LIN {X 0,Y 418.354,Z 136.374,A -85,B 0,C 180,E1 -10247.385,E2 -10247.385} C_VEL
LIN {X 0,Y 418.34,Z 136.372,A -85,B 0,C 180,E1 -10250.328,E2 -10250.328} C_VEL
LIN {X 0,Y 418.511,Z 136.347,A -85,B 0,C 180,E1 -10252.279,E2 -10252.279} C_VEL
LIN {X 0,Y 418.512,Z 136.351,A -85,B 0,C 180,E1 -10254.217,E2 -10254.217} C_VEL
LIN {X 0,Y 418.543,Z 136.347,A -85,B 0,C 180,E1 -10258.075,E2 -10258.075} C_VEL
LIN {X 0,Y 418.671,Z 136.328,A -85,B 0,C 180,E1 -10260,E2 -10260} C_VEL
LIN {X 0,Y 418.508,Z 136.353,A -85,B 0,C 180,E1 -10262.888,E2 -10262.888} C_VEL
LIN {X 0,Y 418.485,Z 136.356,A -85,B 0,C 180,E1 -10266.751,E2 -10266.751} C_VEL
LIN {X 0,Y 418.339,Z 136.373,A -85,B 0,C 180,E1 -10269.671,E2 -10269.671} C_VEL
LIN {X 0,Y 418.344,Z 136.376,A -85,B 0,C 180,E1 -10273.001,E2 -10273.001} C_VEL
LIN {X 0,Y 418.311,Z 136.381,A -85,B 0,C 180,E1 -10276.735,E2 -10276.735} C_VEL
LIN {X 0,Y 418.269,Z 136.382,A -85,B 0,C 180,E1 -10279.79,E2 -10279.79} C_VEL
LIN {X 0,Y 418.236,Z 136.392,A -85,B 0,C 180,E1 -10282.736,E2 -10282.736} C_VEL
LIN {X 0,Y 418.268,Z 136.387,A -85,B 0,C 180,E1 -10285.904,E2 -10285.904} C_VEL
LIN {X 0,Y 418.262,Z 136.385,A -85,B 0,C 180,E1 -10289.162,E2 -10289.162} C_VEL
LIN {X 0,Y 418.279,Z 136.588,A -85,B 0,C 180,E1 -10291.885,E2 -10291.885} C_VEL
LIN {X 0,Y 419.996,Z 144.56,A -85,B 0,C 180,E1 -10293.806,E2 -10293.806} C_VEL
LIN {X 0,Y 422.177,Z 151.711,A -85,B 0,C 180,E1 -10294.075,E2 -10294.075} C_VEL
LIN {X 0,Y 424.507,Z 162.243,A -85,B 0,C 180,E1 -10294.391,E2 -10294.391} C_VEL
LIN {X 0,Y 423.252,Z 251.811,A -85,B 0,C 180,E1 -10296.015,E2 -10296.015} C_VEL
LIN {X 0,Y 422.853,Z 265.002,A -85,B 0,C 180,E1 -10296.445,E2 -10296.445} C_VEL
LIN {X 0,Y 422.454,Z 276.75,A -85,B 0,C 180,E1 -10297.01,E2 -10297.01} C_VEL
LIN {X 0,Y 421.875,Z 288.685,A -85,B 0,C 180,E1 -10297.778,E2 -10297.778} C_VEL
LIN {X 0,Y 421.216,Z 299.793,A -85,B 0,C 180,E1 -10298.706,E2 -10298.706} C_VEL
LIN {X 0,Y 420.478,Z 309.867,A -85,B 0,C 180,E1 -10299.749,E2 -10299.749} C_VEL
LIN {X 0,Y 419.822,Z 318.462,A -85,B 0,C 180,E1 -10300.838,E2 -10300.838} C_VEL
LIN {X 0,Y 419.17,Z 326.786,A -85,B 0,C 180,E1 -10302.118,E2 -10302.118} C_VEL
LIN {X 0,Y 418.53,Z 334.126,A -85,B 0,C 180,E1 -10303.509,E2 -10303.509} C_VEL
LIN {X 0,Y 418.044,Z 340.71,A -85,B 0,C 180,E1 -10305.083,E2 -10305.083} C_VEL
LIN {X 0,Y 417.75,Z 345.057,A -85,B 0,C 180,E1 -10306.389,E2 -10306.389} C_VEL
LIN {X 0,Y 417.461,Z 348.727,A -85,B 0,C 180,E1 -10307.795,E2 -10307.795} C_VEL
LIN {X 0,Y 417.221,Z 351.572,A -85,B 0,C 180,E1 -10309.289,E2 -10309.289} C_VEL
LIN {X 0,Y 417.092,Z 353.429,A -85,B 0,C 180,E1 -10310.814,E2 -10310.814} C_VEL
LIN {X 0,Y 417.018,Z 354.326,A -85,B 0,C 180,E1 -10312.649,E2 -10312.649} C_VEL
LIN {X 0,Y 417.039,Z 354.081,A -85,B 0,C 180,E1 -10313.989,E2 -10313.989} C_VEL
LIN {X 0,Y 417.104,Z 352.704,A -85,B 0,C 180,E1 -10315.652,E2 -10315.652} C_VEL
LIN {X 0,Y 417.278,Z 349.985,A -85,B 0,C 180,E1 -10317.387,E2 -10317.387} C_VEL
LIN {X 0,Y 417.563,Z 345.808,A -85,B 0,C 180,E1 -10319.135,E2 -10319.135} C_VEL
LIN {X 0,Y 417.947,Z 340.265,A -85,B 0,C 180,E1 -10320.814,E2 -10320.814} C_VEL
LIN {X 0,Y 418.428,Z 333.293,A -85,B 0,C 180,E1 -10322.444,E2 -10322.444} C_VEL
LIN {X 0,Y 418.96,Z 325.522,A -85,B 0,C 180,E1 -10323.875,E2 -10323.875} C_VEL
LIN {X 0,Y 419.599,Z 316.285,A -85,B 0,C 180,E1 -10325.246,E2 -10325.246} C_VEL
LIN {X 0,Y 420.213,Z 307.278,A -85,B 0,C 180,E1 -10326.335,E2 -10326.335} C_VEL
LIN {X 0,Y 420.843,Z 297.324,A -85,B 0,C 180,E1 -10327.321,E2 -10327.321} C_VEL
LIN {X 0,Y 421.442,Z 285.916,A -85,B 0,C 180,E1 -10328.22,E2 -10328.22} C_VEL
LIN {X 0,Y 421.997,Z 273.068,A -85,B 0,C 180,E1 -10328.997,E2 -10328.997} C_VEL
LIN {X 0,Y 422.427,Z 260.281,A -85,B 0,C 180,E1 -10329.551,E2 -10329.551} C_VEL
LIN {X 0,Y 422.746,Z 246.227,A -85,B 0,C 180,E1 -10329.932,E2 -10329.932} C_VEL
LIN {X 0,Y 423.437,Z 190.42,A -85,B 0,C 180,E1 -10330.915,E2 -10330.915} C_VEL
LIN {X 0,Y 422.55,Z 182.716,A -85,B 0,C 180,E1 -10331.093,E2 -10331.093} C_VEL
LIN {X 0,Y 418.279,Z 167.8,A -85,B 0,C 180,E1 -10331.551,E2 -10331.551} C_VEL
LIN {X 0,Y 416.448,Z 160.229,A -85,B 0,C 180,E1 -10331.772,E2 -10331.772} C_VEL
LIN {X 0,Y 413.37,Z 146.655,A -85,B 0,C 180,E1 -10332.164,E2 -10332.164} C_VEL
LIN {X 0,Y 412.534,Z 143.848,A -85,B 0,C 180,E1 -10332.276,E2 -10332.276} C_VEL
LIN {X 0,Y 411.31,Z 137.253,A -85,B 0,C 180,E1 -10333.879,E2 -10333.879} C_VEL
LIN {X 0,Y 411.303,Z 137.253,A -85,B 0,C 180,E1 -10337.166,E2 -10337.166} C_VEL
LIN {X 0,Y 411.292,Z 137.25,A -85,B 0,C 180,E1 -10340.161,E2 -10340.161} C_VEL
LIN {X 0,Y 411.452,Z 137.232,A -85,B 0,C 180,E1 -10343.133,E2 -10343.133} C_VEL
LIN {X 0,Y 411.308,Z 137.25,A -85,B 0,C 180,E1 -10345.099,E2 -10345.099} C_VEL
LIN {X 0,Y 411.51,Z 137.222,A -85,B 0,C 180,E1 -10348.043,E2 -10348.043} C_VEL
LIN {X 0,Y 411.64,Z 137.206,A -85,B 0,C 180,E1 -10350,E2 -10350} C_VEL
LIN {X 0,Y 411.457,Z 137.231,A -85,B 0,C 180,E1 -10352.937,E2 -10352.937} C_VEL
LIN {X 0,Y 411.424,Z 137.236,A -85,B 0,C 180,E1 -10356.868,E2 -10356.868} C_VEL
LIN {X 0,Y 411.291,Z 137.249,A -85,B 0,C 180,E1 -10359.839,E2 -10359.839} C_VEL
LIN {X 0,Y 411.305,Z 137.253,A -85,B 0,C 180,E1 -10363.104,E2 -10363.104} C_VEL
LIN {X 0,Y 411.257,Z 137.26,A -85,B 0,C 180,E1 -10366.889,E2 -10366.889} C_VEL
LIN {X 0,Y 411.23,Z 137.257,A -85,B 0,C 180,E1 -10369.987,E2 -10369.987} C_VEL
LIN {X 0,Y 411.196,Z 137.264,A -85,B 0,C 180,E1 -10373.148,E2 -10373.148} C_VEL
LIN {X 0,Y 411.236,Z 137.259,A -85,B 0,C 180,E1 -10376.381,E2 -10376.381} C_VEL
LIN {X 0,Y 411.199,Z 137.26,A -85,B 0,C 180,E1 -10379.713,E2 -10379.713} C_VEL
LIN {X 0,Y 411.205,Z 137.261,A -85,B 0,C 180,E1 -10383.156,E2 -10383.156} C_VEL
LIN {X 0,Y 411.191,Z 137.267,A -85,B 0,C 180,E1 -10386.552,E2 -10386.552} C_VEL
LIN {X 0,Y 411.207,Z 137.26,A -85,B 0,C 180,E1 -10389.727,E2 -10389.727} C_VEL
LIN {X 0,Y 411.172,Z 137.264,A -85,B 0,C 180,E1 -10393.134,E2 -10393.134} C_VEL
LIN {X 0,Y 411.168,Z 137.268,A -85,B 0,C 180,E1 -10395.881,E2 -10395.881} C_VEL
LIN {X 0,Y 411.163,Z 137.266,A -85,B 0,C 180,E1 -10398.771,E2 -10398.771} C_VEL
LIN {X 0,Y 411.21,Z 137.263,A -85,B 0,C 180,E1 -10401.83,E2 -10401.83} C_VEL
LIN {X 0,Y 411.209,Z 137.259,A -85,B 0,C 180,E1 -10405.121,E2 -10405.121} C_VEL
LIN {X 0,Y 411.164,Z 137.271,A -85,B 0,C 180,E1 -10408.003,E2 -10408.003} C_VEL
LIN {X 0,Y 411.216,Z 137.261,A -85,B 0,C 180,E1 -10411.41,E2 -10411.41} C_VEL
LIN {X 0,Y 411.235,Z 137.261,A -85,B 0,C 180,E1 -10413.619,E2 -10413.619} C_VEL
LIN {X 0,Y 411.194,Z 137.261,A -85,B 0,C 180,E1 -10416.852,E2 -10416.852} C_VEL
LIN {X 0,Y 411.213,Z 137.261,A -85,B 0,C 180,E1 -10420.05,E2 -10420.05} C_VEL
LIN {X 0,Y 411.261,Z 137.255,A -85,B 0,C 180,E1 -10423.131,E2 -10423.131} C_VEL
LIN {X 0,Y 411.304,Z 137.249,A -85,B 0,C 180,E1 -10426.896,E2 -10426.896} C_VEL
LIN {X 0,Y 411.292,Z 137.249,A -85,B 0,C 180,E1 -10430.161,E2 -10430.161} C_VEL
LIN {X 0,Y 411.459,Z 137.233,A -85,B 0,C 180,E1 -10433.133,E2 -10433.133} C_VEL
LIN {X 0,Y 411.31,Z 137.252,A -85,B 0,C 180,E1 -10435.099,E2 -10435.099} C_VEL
LIN {X 0,Y 411.512,Z 137.221,A -85,B 0,C 180,E1 -10438.043,E2 -10438.043} C_VEL
LIN {X 0,Y 411.641,Z 137.205,A -85,B 0,C 180,E1 -10440,E2 -10440} C_VEL
LIN {X 0,Y 411.464,Z 137.233,A -85,B 0,C 180,E1 -10442.937,E2 -10442.937} C_VEL
LIN {X 0,Y 411.45,Z 137.235,A -85,B 0,C 180,E1 -10446.867,E2 -10446.867} C_VEL
LIN {X 0,Y 411.292,Z 137.249,A -85,B 0,C 180,E1 -10449.839,E2 -10449.839} C_VEL
LIN {X 0,Y 411.304,Z 137.251,A -85,B 0,C 180,E1 -10453.104,E2 -10453.104} C_VEL
LIN {X 0,Y 411.256,Z 137.258,A -85,B 0,C 180,E1 -10456.889,E2 -10456.889} C_VEL
LIN {X 0,Y 411.23,Z 137.258,A -85,B 0,C 180,E1 -10459.987,E2 -10459.987} C_VEL
LIN {X 0,Y 411.196,Z 137.262,A -85,B 0,C 180,E1 -10463.148,E2 -10463.148} C_VEL
LIN {X 0,Y 411.237,Z 137.262,A -85,B 0,C 180,E1 -10466.381,E2 -10466.381} C_VEL
LIN {X 0,Y 411.2,Z 137.261,A -85,B 0,C 180,E1 -10469.713,E2 -10469.713} C_VEL
LIN {X 0,Y 411.206,Z 137.26,A -85,B 0,C 180,E1 -10473.156,E2 -10473.156} C_VEL
LIN {X 0,Y 411.195,Z 137.264,A -85,B 0,C 180,E1 -10476.553,E2 -10476.553} C_VEL
LIN {X 0,Y 411.227,Z 137.26,A -85,B 0,C 180,E1 -10479.731,E2 -10479.731} C_VEL
LIN {X 0,Y 411.178,Z 137.263,A -85,B 0,C 180,E1 -10483.133,E2 -10483.133} C_VEL
LIN {X 0,Y 411.169,Z 137.27,A -85,B 0,C 180,E1 -10485.881,E2 -10485.881} C_VEL
LIN {X 0,Y 411.201,Z 137.26,A -85,B 0,C 180,E1 -10488.766,E2 -10488.766} C_VEL
LIN {X 0,Y 411.205,Z 137.264,A -85,B 0,C 180,E1 -10492.028,E2 -10492.028} C_VEL
LIN {X 0,Y 411.208,Z 137.266,A -85,B 0,C 180,E1 -10495.667,E2 -10495.667} C_VEL
LIN {X 0,Y 411.191,Z 137.264,A -85,B 0,C 180,E1 -10499.153,E2 -10499.153} C_VEL
LIN {X 0,Y 411.287,Z 137.341,A -85,B 0,C 180,E1 -10501.234,E2 -10501.234} C_VEL
LIN {X 0,Y 413.809,Z 149.635,A -85,B 0,C 180,E1 -10503.796,E2 -10503.796} C_VEL
LIN {X 0,Y 414.551,Z 154.098,A -85,B 0,C 180,E1 -10504.698,E2 -10504.698} C_VEL
LIN {X 0,Y 413.345,Z 171.886,A -85,B 0,C 180,E1 -10508.034,E2 -10508.034} C_VEL
LIN {X 0,Y 412.497,Z 186.557,A -85,B 0,C 180,E1 -10510.757,E2 -10510.757} C_VEL
LIN {X 0,Y 416.517,Z 216.408,A -85,B 0,C 180,E1 -10511.49,E2 -10511.49} C_VEL
LIN {X 0,Y 415.495,Z 295.911,A -85,B 0,C 180,E1 -10512.941,E2 -10512.941} C_VEL
LIN {X 0,Y 414.943,Z 309.622,A -85,B 0,C 180,E1 -10513.392,E2 -10513.392} C_VEL
LIN {X 0,Y 414.318,Z 322.023,A -85,B 0,C 180,E1 -10514,E2 -10514} C_VEL
LIN {X 0,Y 413.48,Z 334.717,A -85,B 0,C 180,E1 -10514.851,E2 -10514.851} C_VEL
LIN {X 0,Y 412.731,Z 346.038,A -85,B 0,C 180,E1 -10515.831,E2 -10515.831} C_VEL
LIN {X 0,Y 411.983,Z 356.552,A -85,B 0,C 180,E1 -10516.977,E2 -10516.977} C_VEL
LIN {X 0,Y 411.43,Z 365.442,A -85,B 0,C 180,E1 -10518.172,E2 -10518.172} C_VEL
LIN {X 0,Y 410.734,Z 374.404,A -85,B 0,C 180,E1 -10519.65,E2 -10519.65} C_VEL
LIN {X 0,Y 410.366,Z 381.605,A -85,B 0,C 180,E1 -10521.133,E2 -10521.133} C_VEL
LIN {X 0,Y 410.171,Z 387.34,A -85,B 0,C 180,E1 -10522.617,E2 -10522.617} C_VEL
LIN {X 0,Y 410.003,Z 391.842,A -85,B 0,C 180,E1 -10524.097,E2 -10524.097} C_VEL
LIN {X 0,Y 410.066,Z 394.22,A -85,B 0,C 180,E1 -10525.084,E2 -10525.084} C_VEL
LIN {X 0,Y 409.974,Z 396.148,A -85,B 0,C 180,E1 -10526.068,E2 -10526.068} C_VEL
LIN {X 0,Y 410.06,Z 397.644,A -85,B 0,C 180,E1 -10527.053,E2 -10527.053} C_VEL
LIN {X 0,Y 410.053,Z 398.68,A -85,B 0,C 180,E1 -10528.036,E2 -10528.036} C_VEL
LIN {X 0,Y 410.033,Z 399.317,A -85,B 0,C 180,E1 -10529.018,E2 -10529.018} C_VEL
LIN {X 0,Y 410.034,Z 399.56,A -85,B 0,C 180,E1 -10530,E2 -10530} C_VEL
LIN {X 0,Y 410.02,Z 399.386,A -85,B 0,C 180,E1 -10530.982,E2 -10530.982} C_VEL
LIN {X 0,Y 410.044,Z 398.781,A -85,B 0,C 180,E1 -10531.964,E2 -10531.964} C_VEL
LIN {X 0,Y 410.029,Z 397.777,A -85,B 0,C 180,E1 -10532.947,E2 -10532.947} C_VEL
LIN {X 0,Y 409.972,Z 396.368,A -85,B 0,C 180,E1 -10533.932,E2 -10533.932} C_VEL
LIN {X 0,Y 410.017,Z 393.411,A -85,B 0,C 180,E1 -10535.409,E2 -10535.409} C_VEL
LIN {X 0,Y 410.078,Z 389.406,A -85,B 0,C 180,E1 -10536.89,E2 -10536.89} C_VEL
LIN {X 0,Y 410.357,Z 383.275,A -85,B 0,C 180,E1 -10538.619,E2 -10538.619} C_VEL
LIN {X 0,Y 410.711,Z 376.554,A -85,B 0,C 180,E1 -10540.102,E2 -10540.102} C_VEL
LIN {X 0,Y 411.339,Z 368.229,A -85,B 0,C 180,E1 -10541.581,E2 -10541.581} C_VEL
LIN {X 0,Y 411.91,Z 359.73,A -85,B 0,C 180,E1 -10542.815,E2 -10542.815} C_VEL
LIN {X 0,Y 412.688,Z 349.532,A -85,B 0,C 180,E1 -10544.019,E2 -10544.019} C_VEL
LIN {X 0,Y 413.565,Z 337.56,A -85,B 0,C 180,E1 -10545.146,E2 -10545.146} C_VEL
LIN {X 0,Y 414.45,Z 325.957,A -85,B 0,C 180,E1 -10545.995,E2 -10545.995} C_VEL
LIN {X 0,Y 415.255,Z 312.671,A -85,B 0,C 180,E1 -10546.721,E2 -10546.721} C_VEL
LIN {X 0,Y 415.952,Z 299.229,A -85,B 0,C 180,E1 -10547.23,E2 -10547.23} C_VEL
LIN {X 0,Y 416.316,Z 284.215,A -85,B 0,C 180,E1 -10547.563,E2 -10547.563} C_VEL
LIN {X 0,Y 417.118,Z 215.058,A -85,B 0,C 180,E1 -10548.823,E2 -10548.823} C_VEL
LIN {X 0,Y 414.02,Z 193.054,A -85,B 0,C 180,E1 -10549.4,E2 -10549.4} C_VEL
LIN {X 0,Y 412.69,Z 185.111,A -85,B 0,C 180,E1 -10549.628,E2 -10549.628} C_VEL
LIN {X 0,Y 413.943,Z 164.842,A -85,B 0,C 180,E1 -10553.381,E2 -10553.381} C_VEL
LIN {X 0,Y 414.609,Z 153.401,A -85,B 0,C 180,E1 -10555.534,E2 -10555.534} C_VEL
LIN {X 0,Y 412.265,Z 141.515,A -85,B 0,C 180,E1 -10558.008,E2 -10558.008} C_VEL
LIN {X 0,Y 411.236,Z 137.263,A -85,B 0,C 180,E1 -10558.951,E2 -10558.951} C_VEL
LIN {X 0,Y 411.167,Z 137.271,A -85,B 0,C 180,E1 -10561.997,E2 -10561.997} C_VEL
LIN {X 0,Y 411.212,Z 137.264,A -85,B 0,C 180,E1 -10564.878,E2 -10564.878} C_VEL
LIN {X 0,Y 411.215,Z 137.27,A -85,B 0,C 180,E1 -10568.17,E2 -10568.17} C_VEL
LIN {X 0,Y 411.201,Z 137.264,A -85,B 0,C 180,E1 -10571.234,E2 -10571.234} C_VEL
LIN {X 0,Y 411.176,Z 137.27,A -85,B 0,C 180,E1 -10574.49,E2 -10574.49} C_VEL
LIN {X 0,Y 411.198,Z 137.264,A -85,B 0,C 180,E1 -10578.197,E2 -10578.197} C_VEL
LIN {X 0,Y 411.23,Z 137.256,A -85,B 0,C 180,E1 -10580.777,E2 -10580.777} C_VEL
LIN {X 0,Y 411.198,Z 137.262,A -85,B 0,C 180,E1 -10584.471,E2 -10584.471} C_VEL
LIN {X 0,Y 411.206,Z 137.258,A -85,B 0,C 180,E1 -10586.873,E2 -10586.873} C_VEL
LIN {X 0,Y 411.232,Z 137.253,A -85,B 0,C 180,E1 -10590.644,E2 -10590.644} C_VEL
LIN {X 0,Y 411.235,Z 137.257,A -85,B 0,C 180,E1 -10593.619,E2 -10593.619} C_VEL
LIN {X 0,Y 411.194,Z 137.26,A -85,B 0,C 180,E1 -10596.852,E2 -10596.852} C_VEL
LIN {X 0,Y 411.214,Z 137.257,A -85,B 0,C 180,E1 -10600.05,E2 -10600.05} C_VEL
LIN {X 0,Y 411.262,Z 137.255,A -85,B 0,C 180,E1 -10603.131,E2 -10603.131} C_VEL
LIN {X 0,Y 411.304,Z 137.25,A -85,B 0,C 180,E1 -10606.896,E2 -10606.896} C_VEL
LIN {X 0,Y 411.292,Z 137.25,A -85,B 0,C 180,E1 -10610.161,E2 -10610.161} C_VEL
LIN {X 0,Y 411.459,Z 137.229,A -85,B 0,C 180,E1 -10613.133,E2 -10613.133} C_VEL
LIN {X 0,Y 411.309,Z 137.251,A -85,B 0,C 180,E1 -10615.099,E2 -10615.099} C_VEL
LIN {X 0,Y 411.512,Z 137.223,A -85,B 0,C 180,E1 -10618.042,E2 -10618.042} C_VEL
LIN {X 0,Y 411.64,Z 137.204,A -85,B 0,C 180,E1 -10620,E2 -10620} C_VEL
LIN {X 0,Y 411.463,Z 137.23,A -85,B 0,C 180,E1 -10622.937,E2 -10622.937} C_VEL
LIN {X 0,Y 411.449,Z 137.233,A -85,B 0,C 180,E1 -10626.867,E2 -10626.867} C_VEL
LIN {X 0,Y 411.291,Z 137.251,A -85,B 0,C 180,E1 -10629.839,E2 -10629.839} C_VEL
LIN {X 0,Y 411.303,Z 137.252,A -85,B 0,C 180,E1 -10633.104,E2 -10633.104} C_VEL
LIN {X 0,Y 411.255,Z 137.26,A -85,B 0,C 180,E1 -10636.889,E2 -10636.889} C_VEL
LIN {X 0,Y 411.228,Z 137.26,A -85,B 0,C 180,E1 -10639.987,E2 -10639.987} C_VEL
LIN {X 0,Y 411.201,Z 137.268,A -85,B 0,C 180,E1 -10643.147,E2 -10643.147} C_VEL
LIN {X 0,Y 411.236,Z 137.262,A -85,B 0,C 180,E1 -10646.381,E2 -10646.381} C_VEL
LIN {X 0,Y 411.198,Z 137.264,A -85,B 0,C 180,E1 -10649.713,E2 -10649.713} C_VEL
LIN {X 0,Y 411.218,Z 137.294,A -85,B 0,C 180,E1 -10651.542,E2 -10651.542} C_VEL
LIN {X 0,Y 412.89,Z 145.086,A -85,B 0,C 180,E1 -10653.449,E2 -10653.449} C_VEL
LIN {X 0,Y 415.599,Z 153.137,A -85,B 0,C 180,E1 -10653.754,E2 -10653.754} C_VEL
LIN {X 0,Y 417.868,Z 163.527,A -85,B 0,C 180,E1 -10654.075,E2 -10654.075} C_VEL
LIN {X 0,Y 416.551,Z 251.828,A -85,B 0,C 180,E1 -10655.699,E2 -10655.699} C_VEL
LIN {X 0,Y 416.127,Z 264.942,A -85,B 0,C 180,E1 -10656.127,E2 -10656.127} C_VEL
LIN {X 0,Y 415.704,Z 277.323,A -85,B 0,C 180,E1 -10656.731,E2 -10656.731} C_VEL
LIN {X 0,Y 415.119,Z 288.673,A -85,B 0,C 180,E1 -10657.469,E2 -10657.469} C_VEL
LIN {X 0,Y 414.391,Z 300.39,A -85,B 0,C 180,E1 -10658.462,E2 -10658.462} C_VEL
LIN {X 0,Y 413.545,Z 311.341,A -85,B 0,C 180,E1 -10659.628,E2 -10659.628} C_VEL
LIN {X 0,Y 412.763,Z 321.03,A -85,B 0,C 180,E1 -10660.926,E2 -10660.926} C_VEL
LIN {X 0,Y 411.924,Z 330.134,A -85,B 0,C 180,E1 -10662.447,E2 -10662.447} C_VEL
LIN {X 0,Y 411.396,Z 336.955,A -85,B 0,C 180,E1 -10663.873,E2 -10663.873} C_VEL
LIN {X 0,Y 410.886,Z 343.002,A -85,B 0,C 180,E1 -10665.47,E2 -10665.47} C_VEL
LIN {X 0,Y 410.609,Z 346.964,A -85,B 0,C 180,E1 -10666.793,E2 -10666.793} C_VEL
LIN {X 0,Y 410.352,Z 349.984,A -85,B 0,C 180,E1 -10668.092,E2 -10668.092} C_VEL
LIN {X 0,Y 410.128,Z 352.203,A -85,B 0,C 180,E1 -10669.37,E2 -10669.37} C_VEL
LIN {X 0,Y 410.036,Z 353.731,A -85,B 0,C 180,E1 -10670.641,E2 -10670.641} C_VEL
LIN {X 0,Y 409.945,Z 354.612,A -85,B 0,C 180,E1 -10672.056,E2 -10672.056} C_VEL
LIN {X 0,Y 409.94,Z 354.611,A -85,B 0,C 180,E1 -10673.684,E2 -10673.684} C_VEL
LIN {X 0,Y 410.014,Z 353.235,A -85,B 0,C 180,E1 -10675.553,E2 -10675.553} C_VEL
LIN {X 0,Y 410.139,Z 350.993,A -85,B 0,C 180,E1 -10677.103,E2 -10677.103} C_VEL
LIN {X 0,Y 410.466,Z 347.088,A -85,B 0,C 180,E1 -10678.881,E2 -10678.881} C_VEL
LIN {X 0,Y 410.717,Z 343.026,A -85,B 0,C 180,E1 -10680.249,E2 -10680.249} C_VEL
LIN {X 0,Y 411.164,Z 336.503,A -85,B 0,C 180,E1 -10681.962,E2 -10681.962} C_VEL
LIN {X 0,Y 411.668,Z 329.487,A -85,B 0,C 180,E1 -10683.404,E2 -10683.404} C_VEL
LIN {X 0,Y 412.306,Z 321.233,A -85,B 0,C 180,E1 -10684.777,E2 -10684.777} C_VEL
LIN {X 0,Y 413.039,Z 311.369,A -85,B 0,C 180,E1 -10686.108,E2 -10686.108} C_VEL
LIN {X 0,Y 413.743,Z 300.579,A -85,B 0,C 180,E1 -10687.267,E2 -10687.267} C_VEL
LIN {X 0,Y 414.469,Z 288.693,A -85,B 0,C 180,E1 -10688.278,E2 -10688.278} C_VEL
LIN {X 0,Y 415.002,Z 277.283,A -85,B 0,C 180,E1 -10689.033,E2 -10689.033} C_VEL
LIN {X 0,Y 415.491,Z 264.693,A -85,B 0,C 180,E1 -10689.647,E2 -10689.647} C_VEL
LIN {X 0,Y 415.811,Z 251.596,A -85,B 0,C 180,E1 -10690.082,E2 -10690.082} C_VEL
LIN {X 0,Y 416.955,Z 162.535,A -85,B 0,C 180,E1 -10691.707,E2 -10691.707} C_VEL
LIN {X 0,Y 416.448,Z 160.229,A -85,B 0,C 180,E1 -10691.772,E2 -10691.772} C_VEL
LIN {X 0,Y 415.218,Z 156.314,A -85,B 0,C 180,E1 -10691.914,E2 -10691.914} C_VEL
LIN {X 0,Y 412.319,Z 151.696,A -85,B 0,C 180,E1 -10692.132,E2 -10692.132} C_VEL
LIN {X 0,Y 406.058,Z 144.867,A -85,B 0,C 180,E1 -10692.558,E2 -10692.558} C_VEL
LIN {X 0,Y 405.256,Z 143.561,A -85,B 0,C 180,E1 -10692.76,E2 -10692.76} C_VEL
LIN {X 0,Y 404.27,Z 138.13,A -85,B 0,C 180,E1 -10694.109,E2 -10694.109} C_VEL
LIN {X 0,Y 404.282,Z 138.126,A -85,B 0,C 180,E1 -10696.939,E2 -10696.939} C_VEL
LIN {X 0,Y 404.257,Z 138.128,A -85,B 0,C 180,E1 -10699.988,E2 -10699.988} C_VEL
LIN {X 0,Y 404.399,Z 138.109,A -85,B 0,C 180,E1 -10703.013,E2 -10703.013} C_VEL
LIN {X 0,Y 404.28,Z 138.124,A -85,B 0,C 180,E1 -10705.014,E2 -10705.014} C_VEL
LIN {X 0,Y 404.479,Z 138.098,A -85,B 0,C 180,E1 -10708.009,E2 -10708.009} C_VEL
LIN {X 0,Y 404.61,Z 138.082,A -85,B 0,C 180,E1 -10710,E2 -10710} C_VEL
LIN {X 0,Y 404.415,Z 138.109,A -85,B 0,C 180,E1 -10712.988,E2 -10712.988} C_VEL
LIN {X 0,Y 404.37,Z 138.116,A -85,B 0,C 180,E1 -10716.988,E2 -10716.988} C_VEL
LIN {X 0,Y 404.257,Z 138.125,A -85,B 0,C 180,E1 -10720.012,E2 -10720.012} C_VEL
LIN {X 0,Y 404.266,Z 138.129,A -85,B 0,C 180,E1 -10723.211,E2 -10723.211} C_VEL
LIN {X 0,Y 404.215,Z 138.136,A -85,B 0,C 180,E1 -10727.007,E2 -10727.007} C_VEL
LIN {X 0,Y 404.163,Z 138.139,A -85,B 0,C 180,E1 -10730.351,E2 -10730.351} C_VEL
LIN {X 0,Y 404.163,Z 138.137,A -85,B 0,C 180,E1 -10733.575,E2 -10733.575} C_VEL
LIN {X 0,Y 404.183,Z 138.134,A -85,B 0,C 180,E1 -10735.766,E2 -10735.766} C_VEL
LIN {X 0,Y 404.195,Z 138.134,A -85,B 0,C 180,E1 -10738,E2 -10738} C_VEL
LIN {X 0,Y 404.138,Z 138.14,A -85,B 0,C 180,E1 -10741.558,E2 -10741.558} C_VEL
LIN {X 0,Y 404.182,Z 138.136,A -85,B 0,C 180,E1 -10745.016,E2 -10745.016} C_VEL
LIN {X 0,Y 404.149,Z 138.141,A -85,B 0,C 180,E1 -10748.757,E2 -10748.757} C_VEL
LIN {X 0,Y 404.121,Z 138.143,A -85,B 0,C 180,E1 -10751.6,E2 -10751.6} C_VEL
LIN {X 0,Y 404.144,Z 138.143,A -85,B 0,C 180,E1 -10754.522,E2 -10754.522} C_VEL
LIN {X 0,Y 404.135,Z 138.14,A -85,B 0,C 180,E1 -10757.296,E2 -10757.296} C_VEL
LIN {X 0,Y 404.167,Z 138.142,A -85,B 0,C 180,E1 -10759.955,E2 -10759.955} C_VEL
LIN {X 0,Y 404.138,Z 138.14,A -85,B 0,C 180,E1 -10763.124,E2 -10763.124} C_VEL
LIN {X 0,Y 404.143,Z 138.143,A -85,B 0,C 180,E1 -10766.188,E2 -10766.188} C_VEL
LIN {X 0,Y 404.144,Z 138.145,A -85,B 0,C 180,E1 -10769.715,E2 -10769.715} C_VEL
LIN {X 0,Y 404.193,Z 138.134,A -85,B 0,C 180,E1 -10773.123,E2 -10773.123} C_VEL
LIN {X 0,Y 404.172,Z 138.138,A -85,B 0,C 180,E1 -10775.334,E2 -10775.334} C_VEL
LIN {X 0,Y 404.136,Z 138.14,A -85,B 0,C 180,E1 -10778.581,E2 -10778.581} C_VEL
LIN {X 0,Y 404.209,Z 138.136,A -85,B 0,C 180,E1 -10781.762,E2 -10781.762} C_VEL
LIN {X 0,Y 404.205,Z 138.133,A -85,B 0,C 180,E1 -10784.882,E2 -10784.882} C_VEL
LIN {X 0,Y 404.255,Z 138.127,A -85,B 0,C 180,E1 -10787.959,E2 -10787.959} C_VEL
LIN {X 0,Y 404.432,Z 138.104,A -85,B 0,C 180,E1 -10792.1,E2 -10792.1} C_VEL
LIN {X 0,Y 404.423,Z 138.105,A -85,B 0,C 180,E1 -10794.015,E2 -10794.015} C_VEL
LIN {X 0,Y 404.481,Z 138.097,A -85,B 0,C 180,E1 -10798.009,E2 -10798.009} C_VEL
LIN {X 0,Y 404.61,Z 138.081,A -85,B 0,C 180,E1 -10800,E2 -10800} C_VEL
LIN {X 0,Y 404.421,Z 138.111,A -85,B 0,C 180,E1 -10802.989,E2 -10802.989} C_VEL
LIN {X 0,Y 404.398,Z 138.114,A -85,B 0,C 180,E1 -10806.988,E2 -10806.988} C_VEL
LIN {X 0,Y 404.257,Z 138.125,A -85,B 0,C 180,E1 -10810.012,E2 -10810.012} C_VEL
LIN {X 0,Y 404.265,Z 138.126,A -85,B 0,C 180,E1 -10813.212,E2 -10813.212} C_VEL
LIN {X 0,Y 404.215,Z 138.134,A -85,B 0,C 180,E1 -10817.007,E2 -10817.007} C_VEL
LIN {X 0,Y 404.163,Z 138.141,A -85,B 0,C 180,E1 -10820.352,E2 -10820.352} C_VEL
LIN {X 0,Y 404.163,Z 138.137,A -85,B 0,C 180,E1 -10823.575,E2 -10823.575} C_VEL
LIN {X 0,Y 404.183,Z 138.135,A -85,B 0,C 180,E1 -10825.767,E2 -10825.767} C_VEL
LIN {X 0,Y 404.195,Z 138.135,A -85,B 0,C 180,E1 -10828,E2 -10828} C_VEL
LIN {X 0,Y 404.139,Z 138.14,A -85,B 0,C 180,E1 -10831.558,E2 -10831.558} C_VEL
LIN {X 0,Y 404.185,Z 138.134,A -85,B 0,C 180,E1 -10835.016,E2 -10835.016} C_VEL
LIN {X 0,Y 404.163,Z 138.138,A -85,B 0,C 180,E1 -10838.756,E2 -10838.756} C_VEL
LIN {X 0,Y 404.15,Z 138.141,A -85,B 0,C 180,E1 -10841.604,E2 -10841.604} C_VEL
LIN {X 0,Y 404.146,Z 138.141,A -85,B 0,C 180,E1 -10844.522,E2 -10844.522} C_VEL
LIN {X 0,Y 404.172,Z 138.137,A -85,B 0,C 180,E1 -10847.301,E2 -10847.301} C_VEL
LIN {X 0,Y 404.17,Z 138.142,A -85,B 0,C 180,E1 -10849.956,E2 -10849.956} C_VEL
LIN {X 0,Y 404.141,Z 138.14,A -85,B 0,C 180,E1 -10853.125,E2 -10853.125} C_VEL
LIN {X 0,Y 404.146,Z 138.143,A -85,B 0,C 180,E1 -10856.188,E2 -10856.188} C_VEL
LIN {X 0,Y 404.147,Z 138.145,A -85,B 0,C 180,E1 -10859.715,E2 -10859.715} C_VEL
LIN {X 0,Y 404.234,Z 138.229,A -85,B 0,C 180,E1 -10860.976,E2 -10860.976} C_VEL
LIN {X 0,Y 406.843,Z 150.891,A -85,B 0,C 180,E1 -10863.664,E2 -10863.664} C_VEL
LIN {X 0,Y 407.579,Z 156.147,A -85,B 0,C 180,E1 -10864.737,E2 -10864.737} C_VEL
LIN {X 0,Y 406.225,Z 175.522,A -85,B 0,C 180,E1 -10868.43,E2 -10868.43} C_VEL
LIN {X 0,Y 405.605,Z 186.046,A -85,B 0,C 180,E1 -10870.417,E2 -10870.417} C_VEL
LIN {X 0,Y 409.694,Z 216.001,A -85,B 0,C 180,E1 -10871.193,E2 -10871.193} C_VEL
LIN {X 0,Y 408.661,Z 295.743,A -85,B 0,C 180,E1 -10872.679,E2 -10872.679} C_VEL
LIN {X 0,Y 408.101,Z 309.38,A -85,B 0,C 180,E1 -10873.138,E2 -10873.138} C_VEL
LIN {X 0,Y 407.403,Z 322.243,A -85,B 0,C 180,E1 -10873.785,E2 -10873.785} C_VEL
LIN {X 0,Y 406.597,Z 334.011,A -85,B 0,C 180,E1 -10874.588,E2 -10874.588} C_VEL
LIN {X 0,Y 405.796,Z 345.389,A -85,B 0,C 180,E1 -10875.584,E2 -10875.584} C_VEL
LIN {X 0,Y 405.014,Z 356.169,A -85,B 0,C 180,E1 -10876.774,E2 -10876.774} C_VEL
LIN {X 0,Y 404.436,Z 364.894,A -85,B 0,C 180,E1 -10877.964,E2 -10877.964} C_VEL
LIN {X 0,Y 403.707,Z 373.886,A -85,B 0,C 180,E1 -10879.468,E2 -10879.468} C_VEL
LIN {X 0,Y 403.314,Z 381.119,A -85,B 0,C 180,E1 -10880.977,E2 -10880.977} C_VEL
LIN {X 0,Y 403.097,Z 386.877,A -85,B 0,C 180,E1 -10882.486,E2 -10882.486} C_VEL
LIN {X 0,Y 402.939,Z 391.399,A -85,B 0,C 180,E1 -10883.993,E2 -10883.993} C_VEL
LIN {X 0,Y 402.968,Z 393.784,A -85,B 0,C 180,E1 -10884.997,E2 -10884.997} C_VEL
LIN {X 0,Y 402.893,Z 395.722,A -85,B 0,C 180,E1 -10885.999,E2 -10885.999} C_VEL
LIN {X 0,Y 402.958,Z 397.23,A -85,B 0,C 180,E1 -10887.001,E2 -10887.001} C_VEL
LIN {X 0,Y 402.982,Z 398.276,A -85,B 0,C 180,E1 -10888.001,E2 -10888.001} C_VEL
LIN {X 0,Y 402.955,Z 398.919,A -85,B 0,C 180,E1 -10889.001,E2 -10889.001} C_VEL
LIN {X 0,Y 402.953,Z 399.168,A -85,B 0,C 180,E1 -10890,E2 -10890} C_VEL
LIN {X 0,Y 402.942,Z 399.005,A -85,B 0,C 180,E1 -10890.999,E2 -10890.999} C_VEL
LIN {X 0,Y 402.973,Z 398.406,A -85,B 0,C 180,E1 -10891.999,E2 -10891.999} C_VEL
LIN {X 0,Y 402.928,Z 397.405,A -85,B 0,C 180,E1 -10892.999,E2 -10892.999} C_VEL
LIN {X 0,Y 402.89,Z 396.001,A -85,B 0,C 180,E1 -10894.001,E2 -10894.001} C_VEL
LIN {X 0,Y 402.909,Z 393.052,A -85,B 0,C 180,E1 -10895.505,E2 -10895.505} C_VEL
LIN {X 0,Y 403.003,Z 389.057,A -85,B 0,C 180,E1 -10897.012,E2 -10897.012} C_VEL
LIN {X 0,Y 403.298,Z 382.944,A -85,B 0,C 180,E1 -10898.771,E2 -10898.771} C_VEL
LIN {X 0,Y 403.681,Z 376.245,A -85,B 0,C 180,E1 -10900.279,E2 -10900.279} C_VEL
LIN {X 0,Y 404.344,Z 367.949,A -85,B 0,C 180,E1 -10901.784,E2 -10901.784} C_VEL
LIN {X 0,Y 404.954,Z 359.485,A -85,B 0,C 180,E1 -10903.039,E2 -10903.039} C_VEL
LIN {X 0,Y 405.834,Z 349.098,A -85,B 0,C 180,E1 -10904.287,E2 -10904.287} C_VEL
LIN {X 0,Y 406.701,Z 337.405,A -85,B 0,C 180,E1 -10905.408,E2 -10905.408} C_VEL
LIN {X 0,Y 407.639,Z 325.888,A -85,B 0,C 180,E1 -10906.27,E2 -10906.27} C_VEL
LIN {X 0,Y 408.468,Z 312.723,A -85,B 0,C 180,E1 -10907.007,E2 -10907.007} C_VEL
LIN {X 0,Y 409.186,Z 299.523,A -85,B 0,C 180,E1 -10907.524,E2 -10907.524} C_VEL
LIN {X 0,Y 409.583,Z 285.061,A -85,B 0,C 180,E1 -10907.861,E2 -10907.861} C_VEL
LIN {X 0,Y 410.462,Z 215.914,A -85,B 0,C 180,E1 -10909.143,E2 -10909.143} C_VEL
LIN {X 0,Y 407.39,Z 194.143,A -85,B 0,C 180,E1 -10909.732,E2 -10909.732} C_VEL
LIN {X 0,Y 405.793,Z 184.674,A -85,B 0,C 180,E1 -10910.01,E2 -10910.01} C_VEL
LIN {X 0,Y 407.039,Z 165.516,A -85,B 0,C 180,E1 -10913.625,E2 -10913.625} C_VEL
LIN {X 0,Y 407.73,Z 155.557,A -85,B 0,C 180,E1 -10915.526,E2 -10915.526} C_VEL
LIN {X 0,Y 406.043,Z 146.16,A -85,B 0,C 180,E1 -10917.503,E2 -10917.503} C_VEL
LIN {X 0,Y 404.209,Z 138.139,A -85,B 0,C 180,E1 -10919.303,E2 -10919.303} C_VEL
LIN {X 0,Y 404.142,Z 138.146,A -85,B 0,C 180,E1 -10922.621,E2 -10922.621} C_VEL
LIN {X 0,Y 404.182,Z 138.139,A -85,B 0,C 180,E1 -10925.19,E2 -10925.19} C_VEL
LIN {X 0,Y 404.164,Z 138.143,A -85,B 0,C 180,E1 -10928.756,E2 -10928.756} C_VEL
LIN {X 0,Y 404.15,Z 138.144,A -85,B 0,C 180,E1 -10931.604,E2 -10931.604} C_VEL
LIN {X 0,Y 404.145,Z 138.146,A -85,B 0,C 180,E1 -10934.522,E2 -10934.522} C_VEL
LIN {X 0,Y 404.171,Z 138.141,A -85,B 0,C 180,E1 -10937.3,E2 -10937.3} C_VEL
LIN {X 0,Y 404.169,Z 138.143,A -85,B 0,C 180,E1 -10939.955,E2 -10939.955} C_VEL
LIN {X 0,Y 404.14,Z 138.142,A -85,B 0,C 180,E1 -10943.124,E2 -10943.124} C_VEL
LIN {X 0,Y 404.144,Z 138.141,A -85,B 0,C 180,E1 -10946.187,E2 -10946.187} C_VEL
LIN {X 0,Y 404.145,Z 138.142,A -85,B 0,C 180,E1 -10949.715,E2 -10949.715} C_VEL
LIN {X 0,Y 404.194,Z 138.135,A -85,B 0,C 180,E1 -10953.123,E2 -10953.123} C_VEL
LIN {X 0,Y 404.173,Z 138.137,A -85,B 0,C 180,E1 -10955.334,E2 -10955.334} C_VEL
LIN {X 0,Y 404.137,Z 138.138,A -85,B 0,C 180,E1 -10958.58,E2 -10958.58} C_VEL
LIN {X 0,Y 404.209,Z 138.132,A -85,B 0,C 180,E1 -10961.762,E2 -10961.762} C_VEL
LIN {X 0,Y 404.205,Z 138.13,A -85,B 0,C 180,E1 -10964.882,E2 -10964.882} C_VEL
LIN {X 0,Y 404.255,Z 138.124,A -85,B 0,C 180,E1 -10967.958,E2 -10967.958} C_VEL
LIN {X 0,Y 404.432,Z 138.101,A -85,B 0,C 180,E1 -10972.099,E2 -10972.099} C_VEL
LIN {X 0,Y 404.423,Z 138.106,A -85,B 0,C 180,E1 -10974.015,E2 -10974.015} C_VEL
LIN {X 0,Y 404.481,Z 138.099,A -85,B 0,C 180,E1 -10978.008,E2 -10978.008} C_VEL
LIN {X 0,Y 404.61,Z 138.079,A -85,B 0,C 180,E1 -10980,E2 -10980} C_VEL
LIN {X 0,Y 404.42,Z 138.107,A -85,B 0,C 180,E1 -10982.988,E2 -10982.988} C_VEL
LIN {X 0,Y 404.397,Z 138.113,A -85,B 0,C 180,E1 -10986.987,E2 -10986.987} C_VEL
LIN {X 0,Y 404.256,Z 138.128,A -85,B 0,C 180,E1 -10990.012,E2 -10990.012} C_VEL
LIN {X 0,Y 404.264,Z 138.128,A -85,B 0,C 180,E1 -10993.211,E2 -10993.211} C_VEL
LIN {X 0,Y 404.213,Z 138.136,A -85,B 0,C 180,E1 -10997.007,E2 -10997.007} C_VEL
LIN {X 0,Y 404.161,Z 138.142,A -85,B 0,C 180,E1 -11000.351,E2 -11000.351} C_VEL
LIN {X 0,Y 404.167,Z 138.143,A -85,B 0,C 180,E1 -11003.574,E2 -11003.574} C_VEL
LIN {X 0,Y 404.181,Z 138.142,A -85,B 0,C 180,E1 -11005.766,E2 -11005.766} C_VEL
LIN {X 0,Y 404.193,Z 138.138,A -85,B 0,C 180,E1 -11008,E2 -11008} C_VEL
LIN {X 0,Y 404.152,Z 138.204,A -85,B 0,C 180,E1 -11011.226,E2 -11011.226} C_VEL
LIN {X 0,Y 405.819,Z 145.686,A -85,B 0,C 180,E1 -11013.06,E2 -11013.06} C_VEL
LIN {X 0,Y 409.283,Z 155.538,A -85,B 0,C 180,E1 -11013.453,E2 -11013.453} C_VEL
LIN {X 0,Y 411.239,Z 165.025,A -85,B 0,C 180,E1 -11013.749,E2 -11013.749} C_VEL
LIN {X 0,Y 409.81,Z 253.323,A -85,B 0,C 180,E1 -11015.414,E2 -11015.414} C_VEL
LIN {X 0,Y 409.365,Z 266.27,A -85,B 0,C 180,E1 -11015.857,E2 -11015.857} C_VEL
LIN {X 0,Y 408.944,Z 278.288,A -85,B 0,C 180,E1 -11016.464,E2 -11016.464} C_VEL
LIN {X 0,Y 408.23,Z 290.688,A -85,B 0,C 180,E1 -11017.309,E2 -11017.309} C_VEL
LIN {X 0,Y 407.503,Z 301.676,A -85,B 0,C 180,E1 -11018.276,E2 -11018.276} C_VEL
LIN {X 0,Y 406.709,Z 311.463,A -85,B 0,C 180,E1 -11019.342,E2 -11019.342} C_VEL
LIN {X 0,Y 405.906,Z 320.945,A -85,B 0,C 180,E1 -11020.619,E2 -11020.619} C_VEL
LIN {X 0,Y 405.129,Z 329.297,A -85,B 0,C 180,E1 -11022.011,E2 -11022.011} C_VEL
LIN {X 0,Y 404.411,Z 337.161,A -85,B 0,C 180,E1 -11023.645,E2 -11023.645} C_VEL
LIN {X 0,Y 403.955,Z 342.57,A -85,B 0,C 180,E1 -11025.064,E2 -11025.064} C_VEL
LIN {X 0,Y 403.608,Z 346.882,A -85,B 0,C 180,E1 -11026.485,E2 -11026.485} C_VEL
LIN {X 0,Y 403.31,Z 350.131,A -85,B 0,C 180,E1 -11027.864,E2 -11027.864} C_VEL
LIN {X 0,Y 402.998,Z 353.317,A -85,B 0,C 180,E1 -11029.816,E2 -11029.816} C_VEL
LIN {X 0,Y 402.891,Z 354.868,A -85,B 0,C 180,E1 -11031.718,E2 -11031.718} C_VEL
LIN {X 0,Y 402.865,Z 355.012,A -85,B 0,C 180,E1 -11033.621,E2 -11033.621} C_VEL
LIN {X 0,Y 402.879,Z 354.125,A -85,B 0,C 180,E1 -11035.073,E2 -11035.073} C_VEL
LIN {X 0,Y 403.053,Z 351.952,A -85,B 0,C 180,E1 -11036.821,E2 -11036.821} C_VEL
LIN {X 0,Y 403.35,Z 348.311,A -85,B 0,C 180,E1 -11038.625,E2 -11038.625} C_VEL
LIN {X 0,Y 403.7,Z 342.895,A -85,B 0,C 180,E1 -11040.51,E2 -11040.51} C_VEL
LIN {X 0,Y 404.097,Z 337.309,A -85,B 0,C 180,E1 -11041.993,E2 -11041.993} C_VEL
LIN {X 0,Y 404.628,Z 330.557,A -85,B 0,C 180,E1 -11043.433,E2 -11043.433} C_VEL
LIN {X 0,Y 405.286,Z 322.25,A -85,B 0,C 180,E1 -11044.859,E2 -11044.859} C_VEL
LIN {X 0,Y 405.994,Z 313.034,A -85,B 0,C 180,E1 -11046.146,E2 -11046.146} C_VEL
LIN {X 0,Y 406.644,Z 303.348,A -85,B 0,C 180,E1 -11047.251,E2 -11047.251} C_VEL
LIN {X 0,Y 407.355,Z 293.182,A -85,B 0,C 180,E1 -11048.189,E2 -11048.189} C_VEL
LIN {X 0,Y 407.964,Z 281.284,A -85,B 0,C 180,E1 -11049.056,E2 -11049.056} C_VEL
LIN {X 0,Y 408.515,Z 268.751,A -85,B 0,C 180,E1 -11049.744,E2 -11049.744} C_VEL
LIN {X 0,Y 408.915,Z 255.775,A -85,B 0,C 180,E1 -11050.241,E2 -11050.241} C_VEL
LIN {X 0,Y 409.219,Z 239.416,A -85,B 0,C 180,E1 -11050.6,E2 -11050.6} C_VEL
LIN {X 0,Y 410.2,Z 163.689,A -85,B 0,C 180,E1 -11051.985,E2 -11051.985} C_VEL
LIN {X 0,Y 406.938,Z 149.062,A -85,B 0,C 180,E1 -11052.413,E2 -11052.413} C_VEL
LIN {X 0,Y 405.377,Z 144.215,A -85,B 0,C 180,E1 -11052.599,E2 -11052.599} C_VEL
LIN {X 0,Y 405.256,Z 143.561,A -85,B 0,C 180,E1 -11052.76,E2 -11052.76} C_VEL
LIN {X 0,Y 404.239,Z 141.814,A -85,B 0,C 180,E1 -11053.252,E2 -11053.252} C_VEL
LIN {X 0,Y 400.972,Z 139.965,A -85,B 0,C 180,E1 -11054.061,E2 -11054.061} C_VEL
LIN {X 0,Y 397.891,Z 139.139,A -85,B 0,C 180,E1 -11054.923,E2 -11054.923} C_VEL
LIN {X 0,Y 397.175,Z 139.013,A -85,B 0,C 180,E1 -11055.493,E2 -11055.493} C_VEL
LIN {X 0,Y 397.198,Z 139.005,A -85,B 0,C 180,E1 -11058.777,E2 -11058.777} C_VEL
LIN {X 0,Y 397.361,Z 138.986,A -85,B 0,C 180,E1 -11062.076,E2 -11062.076} C_VEL
LIN {X 0,Y 397.252,Z 138.999,A -85,B 0,C 180,E1 -11064.925,E2 -11064.925} C_VEL
LIN {X 0,Y 397.448,Z 138.975,A -85,B 0,C 180,E1 -11067.973,E2 -11067.973} C_VEL
LIN {X 0,Y 397.579,Z 138.958,A -85,B 0,C 180,E1 -11070,E2 -11070} C_VEL
LIN {X 0,Y 397.375,Z 138.987,A -85,B 0,C 180,E1 -11073.041,E2 -11073.041} C_VEL
LIN {X 0,Y 397.346,Z 138.986,A -85,B 0,C 180,E1 -11076.092,E2 -11076.092} C_VEL
LIN {X 0,Y 397.236,Z 139.006,A -85,B 0,C 180,E1 -11079.162,E2 -11079.162} C_VEL
LIN {X 0,Y 397.219,Z 139.002,A -85,B 0,C 180,E1 -11082.258,E2 -11082.258} C_VEL
LIN {X 0,Y 397.179,Z 139.009,A -85,B 0,C 180,E1 -11085.392,E2 -11085.392} C_VEL
LIN {X 0,Y 397.158,Z 139.013,A -85,B 0,C 180,E1 -11088.574,E2 -11088.574} C_VEL
LIN {X 0,Y 397.095,Z 139.017,A -85,B 0,C 180,E1 -11091.818,E2 -11091.818} C_VEL
LIN {X 0,Y 397.152,Z 139.01,A -85,B 0,C 180,E1 -11095.512,E2 -11095.512} C_VEL
LIN {X 0,Y 397.122,Z 139.02,A -85,B 0,C 180,E1 -11098.543,E2 -11098.543} C_VEL
LIN {X 0,Y 397.077,Z 139.022,A -85,B 0,C 180,E1 -11102.072,E2 -11102.072} C_VEL
LIN {X 0,Y 397.117,Z 139.015,A -85,B 0,C 180,E1 -11105.503,E2 -11105.503} C_VEL
LIN {X 0,Y 397.125,Z 139.015,A -85,B 0,C 180,E1 -11108.861,E2 -11108.861} C_VEL
LIN {X 0,Y 397.068,Z 139.027,A -85,B 0,C 180,E1 -11112.267,E2 -11112.267} C_VEL
LIN {X 0,Y 397.086,Z 139.019,A -85,B 0,C 180,E1 -11115.069,E2 -11115.069} C_VEL
LIN {X 0,Y 397.065,Z 139.026,A -85,B 0,C 180,E1 -11118.021,E2 -11118.021} C_VEL
LIN {X 0,Y 397.132,Z 139.013,A -85,B 0,C 180,E1 -11121.138,E2 -11121.138} C_VEL
LIN {X 0,Y 397.118,Z 139.016,A -85,B 0,C 180,E1 -11124.496,E2 -11124.496} C_VEL
LIN {X 0,Y 397.077,Z 139.026,A -85,B 0,C 180,E1 -11127.929,E2 -11127.929} C_VEL
LIN {X 0,Y 397.12,Z 139.017,A -85,B 0,C 180,E1 -11131.456,E2 -11131.456} C_VEL
LIN {X 0,Y 397.15,Z 139.011,A -85,B 0,C 180,E1 -11134.488,E2 -11134.488} C_VEL
LIN {X 0,Y 397.094,Z 139.019,A -85,B 0,C 180,E1 -11138.182,E2 -11138.182} C_VEL
LIN {X 0,Y 397.161,Z 139.014,A -85,B 0,C 180,E1 -11141.427,E2 -11141.427} C_VEL
LIN {X 0,Y 397.178,Z 139.007,A -85,B 0,C 180,E1 -11144.608,E2 -11144.608} C_VEL
LIN {X 0,Y 397.218,Z 139.005,A -85,B 0,C 180,E1 -11147.742,E2 -11147.742} C_VEL
LIN {X 0,Y 397.393,Z 138.981,A -85,B 0,C 180,E1 -11152.041,E2 -11152.041} C_VEL
LIN {X 0,Y 397.254,Z 139.001,A -85,B 0,C 180,E1 -11154.925,E2 -11154.925} C_VEL
LIN {X 0,Y 397.45,Z 138.973,A -85,B 0,C 180,E1 -11157.974,E2 -11157.974} C_VEL
LIN {X 0,Y 397.579,Z 138.957,A -85,B 0,C 180,E1 -11160,E2 -11160} C_VEL
LIN {X 0,Y 397.379,Z 138.989,A -85,B 0,C 180,E1 -11163.042,E2 -11163.042} C_VEL
LIN {X 0,Y 397.369,Z 138.983,A -85,B 0,C 180,E1 -11166.092,E2 -11166.092} C_VEL
LIN {X 0,Y 397.252,Z 139.001,A -85,B 0,C 180,E1 -11169.162,E2 -11169.162} C_VEL
LIN {X 0,Y 397.218,Z 139.003,A -85,B 0,C 180,E1 -11172.258,E2 -11172.258} C_VEL
LIN {X 0,Y 397.178,Z 139.008,A -85,B 0,C 180,E1 -11175.392,E2 -11175.392} C_VEL
LIN {X 0,Y 397.162,Z 139.015,A -85,B 0,C 180,E1 -11178.574,E2 -11178.574} C_VEL
LIN {X 0,Y 397.095,Z 139.018,A -85,B 0,C 180,E1 -11181.819,E2 -11181.819} C_VEL
LIN {X 0,Y 397.152,Z 139.01,A -85,B 0,C 180,E1 -11185.513,E2 -11185.513} C_VEL
LIN {X 0,Y 397.122,Z 139.019,A -85,B 0,C 180,E1 -11188.544,E2 -11188.544} C_VEL
LIN {X 0,Y 397.078,Z 139.024,A -85,B 0,C 180,E1 -11192.072,E2 -11192.072} C_VEL
LIN {X 0,Y 397.12,Z 139.015,A -85,B 0,C 180,E1 -11195.504,E2 -11195.504} C_VEL
LIN {X 0,Y 397.137,Z 139.013,A -85,B 0,C 180,E1 -11198.863,E2 -11198.863} C_VEL
LIN {X 0,Y 397.114,Z 139.019,A -85,B 0,C 180,E1 -11202.262,E2 -11202.262} C_VEL
LIN {X 0,Y 397.087,Z 139.018,A -85,B 0,C 180,E1 -11205.069,E2 -11205.069} C_VEL
LIN {X 0,Y 397.111,Z 139.021,A -85,B 0,C 180,E1 -11208.014,E2 -11208.014} C_VEL
LIN {X 0,Y 397.138,Z 139.013,A -85,B 0,C 180,E1 -11211.138,E2 -11211.138} C_VEL
LIN {X 0,Y 397.121,Z 139.014,A -85,B 0,C 180,E1 -11214.497,E2 -11214.497} C_VEL
LIN {X 0,Y 397.08,Z 139.023,A -85,B 0,C 180,E1 -11217.929,E2 -11217.929} C_VEL
LIN {X 0,Y 397.171,Z 139.05,A -85,B 0,C 180,E1 -11220.7,E2 -11220.7} C_VEL
LIN {X 0,Y 399.675,Z 150.997,A -85,B 0,C 180,E1 -11223.29,E2 -11223.29} C_VEL
LIN {X 0,Y 400.634,Z 157.005,A -85,B 0,C 180,E1 -11224.546,E2 -11224.546} C_VEL
LIN {X 0,Y 399.236,Z 176.384,A -85,B 0,C 180,E1 -11228.304,E2 -11228.304} C_VEL
LIN {X 0,Y 398.696,Z 185.973,A -85,B 0,C 180,E1 -11230.123,E2 -11230.123} C_VEL
LIN {X 0,Y 402.955,Z 217.73,A -85,B 0,C 180,E1 -11230.935,E2 -11230.935} C_VEL
LIN {X 0,Y 401.837,Z 295.377,A -85,B 0,C 180,E1 -11232.408,E2 -11232.408} C_VEL
LIN {X 0,Y 401.26,Z 309.01,A -85,B 0,C 180,E1 -11232.874,E2 -11232.874} C_VEL
LIN {X 0,Y 400.549,Z 321.364,A -85,B 0,C 180,E1 -11233.5,E2 -11233.5} C_VEL
LIN {X 0,Y 399.722,Z 333.247,A -85,B 0,C 180,E1 -11234.316,E2 -11234.316} C_VEL
LIN {X 0,Y 398.89,Z 344.703,A -85,B 0,C 180,E1 -11235.329,E2 -11235.329} C_VEL
LIN {X 0,Y 398.162,Z 354.524,A -85,B 0,C 180,E1 -11236.41,E2 -11236.41} C_VEL
LIN {X 0,Y 397.43,Z 364.331,A -85,B 0,C 180,E1 -11237.749,E2 -11237.749} C_VEL
LIN {X 0,Y 396.682,Z 373.359,A -85,B 0,C 180,E1 -11239.279,E2 -11239.279} C_VEL
LIN {X 0,Y 396.282,Z 380.63,A -85,B 0,C 180,E1 -11240.816,E2 -11240.816} C_VEL
LIN {X 0,Y 396.03,Z 386.415,A -85,B 0,C 180,E1 -11242.351,E2 -11242.351} C_VEL
LIN {X 0,Y 395.83,Z 391.716,A -85,B 0,C 180,E1 -11244.194,E2 -11244.194} C_VEL
LIN {X 0,Y 395.814,Z 395.296,A -85,B 0,C 180,E1 -11245.927,E2 -11245.927} C_VEL
LIN {X 0,Y 395.858,Z 396.815,A -85,B 0,C 180,E1 -11246.947,E2 -11246.947} C_VEL
LIN {X 0,Y 395.912,Z 397.872,A -85,B 0,C 180,E1 -11247.965,E2 -11247.965} C_VEL
LIN {X 0,Y 395.879,Z 398.521,A -85,B 0,C 180,E1 -11248.983,E2 -11248.983} C_VEL
LIN {X 0,Y 395.875,Z 398.775,A -85,B 0,C 180,E1 -11250,E2 -11250} C_VEL
LIN {X 0,Y 395.868,Z 398.623,A -85,B 0,C 180,E1 -11251.017,E2 -11251.017} C_VEL
LIN {X 0,Y 395.902,Z 398.031,A -85,B 0,C 180,E1 -11252.035,E2 -11252.035} C_VEL
LIN {X 0,Y 395.81,Z 395.638,A -85,B 0,C 180,E1 -11254.073,E2 -11254.073} C_VEL
LIN {X 0,Y 395.801,Z 392.346,A -85,B 0,C 180,E1 -11255.768,E2 -11255.768} C_VEL
LIN {X 0,Y 395.931,Z 388.725,A -85,B 0,C 180,E1 -11257.138,E2 -11257.138} C_VEL
LIN {X 0,Y 396.232,Z 382.64,A -85,B 0,C 180,E1 -11258.928,E2 -11258.928} C_VEL
LIN {X 0,Y 396.654,Z 375.958,A -85,B 0,C 180,E1 -11260.464,E2 -11260.464} C_VEL
LIN {X 0,Y 397.355,Z 367.681,A -85,B 0,C 180,E1 -11261.995,E2 -11261.995} C_VEL
LIN {X 0,Y 398.021,Z 359.241,A -85,B 0,C 180,E1 -11263.27,E2 -11263.27} C_VEL
LIN {X 0,Y 398.939,Z 348.902,A -85,B 0,C 180,E1 -11264.539,E2 -11264.539} C_VEL
LIN {X 0,Y 399.863,Z 337.251,A -85,B 0,C 180,E1 -11265.678,E2 -11265.678} C_VEL
LIN {X 0,Y 400.822,Z 325.806,A -85,B 0,C 180,E1 -11266.554,E2 -11266.554} C_VEL
LIN {X 0,Y 401.608,Z 314.067,A -85,B 0,C 180,E1 -11267.241,E2 -11267.241} C_VEL
LIN {X 0,Y 402.41,Z 300.664,A -85,B 0,C 180,E1 -11267.796,E2 -11267.796} C_VEL
LIN {X 0,Y 402.823,Z 287.637,A -85,B 0,C 180,E1 -11268.138,E2 -11268.138} C_VEL
LIN {X 0,Y 403.757,Z 216.103,A -85,B 0,C 180,E1 -11269.495,E2 -11269.495} C_VEL
LIN {X 0,Y 400.83,Z 195.386,A -85,B 0,C 180,E1 -11270.072,E2 -11270.072} C_VEL
LIN {X 0,Y 398.913,Z 184.244,A -85,B 0,C 180,E1 -11270.409,E2 -11270.409} C_VEL
LIN {X 0,Y 400.215,Z 165.275,A -85,B 0,C 180,E1 -11274.055,E2 -11274.055} C_VEL
LIN {X 0,Y 400.823,Z 156.752,A -85,B 0,C 180,E1 -11275.719,E2 -11275.719} C_VEL
LIN {X 0,Y 398.868,Z 146.269,A -85,B 0,C 180,E1 -11277.977,E2 -11277.977} C_VEL
LIN {X 0,Y 397.129,Z 139.021,A -85,B 0,C 180,E1 -11279.631,E2 -11279.631} C_VEL
LIN {X 0,Y 397.116,Z 139.02,A -85,B 0,C 180,E1 -11283.272,E2 -11283.272} C_VEL
LIN {X 0,Y 397.11,Z 139.021,A -85,B 0,C 180,E1 -11285.734,E2 -11285.734} C_VEL
LIN {X 0,Y 397.117,Z 139.021,A -85,B 0,C 180,E1 -11289.576,E2 -11289.576} C_VEL
LIN {X 0,Y 397.114,Z 139.025,A -85,B 0,C 180,E1 -11292.261,E2 -11292.261} C_VEL
LIN {X 0,Y 397.087,Z 139.023,A -85,B 0,C 180,E1 -11295.068,E2 -11295.068} C_VEL
LIN {X 0,Y 397.11,Z 139.02,A -85,B 0,C 180,E1 -11298.014,E2 -11298.014} C_VEL
LIN {X 0,Y 397.136,Z 139.012,A -85,B 0,C 180,E1 -11301.137,E2 -11301.137} C_VEL
LIN {X 0,Y 397.119,Z 139.016,A -85,B 0,C 180,E1 -11304.496,E2 -11304.496} C_VEL
LIN {X 0,Y 397.078,Z 139.024,A -85,B 0,C 180,E1 -11307.928,E2 -11307.928} C_VEL
LIN {X 0,Y 397.121,Z 139.015,A -85,B 0,C 180,E1 -11311.456,E2 -11311.456} C_VEL
LIN {X 0,Y 397.151,Z 139.008,A -85,B 0,C 180,E1 -11314.487,E2 -11314.487} C_VEL
LIN {X 0,Y 397.094,Z 139.017,A -85,B 0,C 180,E1 -11318.181,E2 -11318.181} C_VEL
LIN {X 0,Y 397.161,Z 139.008,A -85,B 0,C 180,E1 -11321.426,E2 -11321.426} C_VEL
LIN {X 0,Y 397.178,Z 139.004,A -85,B 0,C 180,E1 -11324.608,E2 -11324.608} C_VEL
LIN {X 0,Y 397.218,Z 139.002,A -85,B 0,C 180,E1 -11327.742,E2 -11327.742} C_VEL
LIN {X 0,Y 397.393,Z 138.978,A -85,B 0,C 180,E1 -11332.041,E2 -11332.041} C_VEL
LIN {X 0,Y 397.253,Z 139.003,A -85,B 0,C 180,E1 -11334.925,E2 -11334.925} C_VEL
LIN {X 0,Y 397.449,Z 138.975,A -85,B 0,C 180,E1 -11337.973,E2 -11337.973} C_VEL
LIN {X 0,Y 397.579,Z 138.955,A -85,B 0,C 180,E1 -11340,E2 -11340} C_VEL
LIN {X 0,Y 397.379,Z 138.984,A -85,B 0,C 180,E1 -11343.041,E2 -11343.041} C_VEL
LIN {X 0,Y 397.343,Z 138.987,A -85,B 0,C 180,E1 -11346.567,E2 -11346.567} C_VEL
LIN {X 0,Y 397.251,Z 139.002,A -85,B 0,C 180,E1 -11349.162,E2 -11349.162} C_VEL
LIN {X 0,Y 397.217,Z 139.004,A -85,B 0,C 180,E1 -11352.258,E2 -11352.258} C_VEL
LIN {X 0,Y 397.177,Z 139.01,A -85,B 0,C 180,E1 -11355.392,E2 -11355.392} C_VEL
LIN {X 0,Y 397.16,Z 139.014,A -85,B 0,C 180,E1 -11358.573,E2 -11358.573} C_VEL
LIN {X 0,Y 397.094,Z 139.02,A -85,B 0,C 180,E1 -11361.818,E2 -11361.818} C_VEL
LIN {X 0,Y 397.154,Z 139.018,A -85,B 0,C 180,E1 -11365.132,E2 -11365.132} C_VEL
LIN {X 0,Y 397.16,Z 139.016,A -85,B 0,C 180,E1 -11367.776,E2 -11367.776} C_VEL
LIN {X 0,Y 397.124,Z 139.042,A -85,B 0,C 180,E1 -11370.878,E2 -11370.878} C_VEL
LIN {X 0,Y 398.647,Z 145.968,A -85,B 0,C 180,E1 -11372.639,E2 -11372.639} C_VEL
LIN {X 0,Y 402.845,Z 157.415,A -85,B 0,C 180,E1 -11373.122,E2 -11373.122} C_VEL
LIN {X 0,Y 404.638,Z 165.443,A -85,B 0,C 180,E1 -11373.386,E2 -11373.386} C_VEL
LIN {X 0,Y 403.142,Z 253.262,A -85,B 0,C 180,E1 -11375.071,E2 -11375.071} C_VEL
LIN {X 0,Y 402.685,Z 266.525,A -85,B 0,C 180,E1 -11375.53,E2 -11375.53} C_VEL
LIN {X 0,Y 402.209,Z 278.432,A -85,B 0,C 180,E1 -11376.138,E2 -11376.138} C_VEL
LIN {X 0,Y 401.478,Z 290.868,A -85,B 0,C 180,E1 -11376.995,E2 -11376.995} C_VEL
LIN {X 0,Y 400.686,Z 302.262,A -85,B 0,C 180,E1 -11378.015,E2 -11378.015} C_VEL
LIN {X 0,Y 399.875,Z 311.926,A -85,B 0,C 180,E1 -11379.088,E2 -11379.088} C_VEL
LIN {X 0,Y 399.009,Z 321.36,A -85,B 0,C 180,E1 -11380.379,E2 -11380.379} C_VEL
LIN {X 0,Y 398.206,Z 329.648,A -85,B 0,C 180,E1 -11381.783,E2 -11381.783} C_VEL
LIN {X 0,Y 397.507,Z 336.363,A -85,B 0,C 180,E1 -11383.176,E2 -11383.176} C_VEL
LIN {X 0,Y 396.947,Z 343.019,A -85,B 0,C 180,E1 -11384.911,E2 -11384.911} C_VEL
LIN {X 0,Y 396.514,Z 347.972,A -85,B 0,C 180,E1 -11386.61,E2 -11386.61} C_VEL
LIN {X 0,Y 396.18,Z 351.343,A -85,B 0,C 180,E1 -11388.164,E2 -11388.164} C_VEL
LIN {X 0,Y 395.92,Z 353.737,A -85,B 0,C 180,E1 -11389.755,E2 -11389.755} C_VEL
LIN {X 0,Y 395.82,Z 355.221,A -85,B 0,C 180,E1 -11391.579,E2 -11391.579} C_VEL
LIN {X 0,Y 395.777,Z 355.508,A -85,B 0,C 180,E1 -11393.043,E2 -11393.043} C_VEL
LIN {X 0,Y 395.799,Z 354.771,A -85,B 0,C 180,E1 -11394.765,E2 -11394.765} C_VEL
LIN {X 0,Y 395.949,Z 352.694,A -85,B 0,C 180,E1 -11396.617,E2 -11396.617} C_VEL
LIN {X 0,Y 396.213,Z 349.463,A -85,B 0,C 180,E1 -11398.366,E2 -11398.366} C_VEL
LIN {X 0,Y 396.589,Z 344.388,A -85,B 0,C 180,E1 -11400.265,E2 -11400.265} C_VEL
LIN {X 0,Y 396.982,Z 338.669,A -85,B 0,C 180,E1 -11401.877,E2 -11401.877} C_VEL
LIN {X 0,Y 397.599,Z 331.405,A -85,B 0,C 180,E1 -11403.492,E2 -11403.492} C_VEL
LIN {X 0,Y 398.257,Z 323.228,A -85,B 0,C 180,E1 -11404.943,E2 -11404.943} C_VEL
LIN {X 0,Y 399.046,Z 313.577,A -85,B 0,C 180,E1 -11406.323,E2 -11406.323} C_VEL
LIN {X 0,Y 399.765,Z 303.239,A -85,B 0,C 180,E1 -11407.52,E2 -11407.52} C_VEL
LIN {X 0,Y 400.601,Z 291.893,A -85,B 0,C 180,E1 -11408.555,E2 -11408.555} C_VEL
LIN {X 0,Y 401.231,Z 279.709,A -85,B 0,C 180,E1 -11409.426,E2 -11409.426} C_VEL
LIN {X 0,Y 401.744,Z 268.03,A -85,B 0,C 180,E1 -11410.055,E2 -11410.055} C_VEL
LIN {X 0,Y 402.118,Z 255.609,A -85,B 0,C 180,E1 -11410.523,E2 -11410.523} C_VEL
LIN {X 0,Y 402.4,Z 239.693,A -85,B 0,C 180,E1 -11410.876,E2 -11410.876} C_VEL
LIN {X 0,Y 403.394,Z 164.368,A -85,B 0,C 180,E1 -11412.283,E2 -11412.283} C_VEL
LIN {X 0,Y 400.467,Z 151.334,A -85,B 0,C 180,E1 -11412.675,E2 -11412.675} C_VEL
LIN {X 0,Y 398.242,Z 144.562,A -85,B 0,C 180,E1 -11412.939,E2 -11412.939} C_VEL
LIN {X 0,Y 397.215,Z 139.007,A -85,B 0,C 180,E1 -11414.347,E2 -11414.347} C_VEL
LIN {X 0,Y 397.175,Z 139.013,A -85,B 0,C 180,E1 -11415.493,E2 -11415.493} C_VEL
LIN {X 0,Y 396.523,Z 139.1,A -85,B 0,C 180,E1 -11416.339,E2 -11416.339} C_VEL
LIN {X 0,Y 393.677,Z 139.458,A -85,B 0,C 180,E1 -11417.715,E2 -11417.715} C_VEL
LIN {X 0,Y 391.267,Z 139.754,A -85,B 0,C 180,E1 -11418.827,E2 -11418.827} C_VEL
LIN {X 0,Y 390.243,Z 139.877,A -85,B 0,C 180,E1 -11419.686,E2 -11419.686} C_VEL
LIN {X 0,Y 390.165,Z 139.883,A -85,B 0,C 180,E1 -11419.977,E2 -11419.977} C_VEL
LIN {X 0,Y 390.301,Z 139.864,A -85,B 0,C 180,E1 -11422.759,E2 -11422.759} C_VEL
LIN {X 0,Y 390.224,Z 139.874,A -85,B 0,C 180,E1 -11424.834,E2 -11424.834} C_VEL
LIN {X 0,Y 390.417,Z 139.851,A -85,B 0,C 180,E1 -11427.937,E2 -11427.937} C_VEL
LIN {X 0,Y 390.548,Z 139.834,A -85,B 0,C 180,E1 -11430,E2 -11430} C_VEL
LIN {X 0,Y 390.309,Z 139.867,A -85,B 0,C 180,E1 -11433.097,E2 -11433.097} C_VEL
LIN {X 0,Y 390.3,Z 139.864,A -85,B 0,C 180,E1 -11436.202,E2 -11436.202} C_VEL
LIN {X 0,Y 390.193,Z 139.881,A -85,B 0,C 180,E1 -11439.329,E2 -11439.329} C_VEL
LIN {X 0,Y 390.171,Z 139.881,A -85,B 0,C 180,E1 -11442.483,E2 -11442.483} C_VEL
LIN {X 0,Y 390.139,Z 139.884,A -85,B 0,C 180,E1 -11445.677,E2 -11445.677} C_VEL
LIN {X 0,Y 390.102,Z 139.895,A -85,B 0,C 180,E1 -11448.922,E2 -11448.922} C_VEL
LIN {X 0,Y 390.037,Z 139.898,A -85,B 0,C 180,E1 -11452.234,E2 -11452.234} C_VEL
LIN {X 0,Y 390.118,Z 139.886,A -85,B 0,C 180,E1 -11455.743,E2 -11455.743} C_VEL
LIN {X 0,Y 390.058,Z 139.896,A -85,B 0,C 180,E1 -11459.109,E2 -11459.109} C_VEL
LIN {X 0,Y 390.041,Z 139.901,A -85,B 0,C 180,E1 -11462.721,E2 -11462.721} C_VEL
LIN {X 0,Y 390.054,Z 139.895,A -85,B 0,C 180,E1 -11465.825,E2 -11465.825} C_VEL
LIN {X 0,Y 390.065,Z 139.893,A -85,B 0,C 180,E1 -11469.218,E2 -11469.218} C_VEL
LIN {X 0,Y 390.041,Z 139.902,A -85,B 0,C 180,E1 -11472.374,E2 -11472.374} C_VEL
LIN {X 0,Y 390.043,Z 139.896,A -85,B 0,C 180,E1 -11475.354,E2 -11475.354} C_VEL
LIN {X 0,Y 390.03,Z 139.904,A -85,B 0,C 180,E1 -11478.187,E2 -11478.187} C_VEL
LIN {X 0,Y 390.091,Z 139.89,A -85,B 0,C 180,E1 -11480.908,E2 -11480.908} C_VEL
LIN {X 0,Y 390.084,Z 139.891,A -85,B 0,C 180,E1 -11484.793,E2 -11484.793} C_VEL
LIN {X 0,Y 390.03,Z 139.904,A -85,B 0,C 180,E1 -11487.875,E2 -11487.875} C_VEL
LIN {X 0,Y 390.056,Z 139.894,A -85,B 0,C 180,E1 -11490.891,E2 -11490.891} C_VEL
LIN {X 0,Y 390.117,Z 139.888,A -85,B 0,C 180,E1 -11494.257,E2 -11494.257} C_VEL
LIN {X 0,Y 390.036,Z 139.902,A -85,B 0,C 180,E1 -11497.766,E2 -11497.766} C_VEL
LIN {X 0,Y 390.104,Z 139.89,A -85,B 0,C 180,E1 -11501.078,E2 -11501.078} C_VEL
LIN {X 0,Y 390.138,Z 139.884,A -85,B 0,C 180,E1 -11504.323,E2 -11504.323} C_VEL
LIN {X 0,Y 390.169,Z 139.886,A -85,B 0,C 180,E1 -11507.517,E2 -11507.517} C_VEL
LIN {X 0,Y 390.313,Z 139.865,A -85,B 0,C 180,E1 -11511.718,E2 -11511.718} C_VEL
LIN {X 0,Y 390.329,Z 139.862,A -85,B 0,C 180,E1 -11513.798,E2 -11513.798} C_VEL
LIN {X 0,Y 390.419,Z 139.849,A -85,B 0,C 180,E1 -11517.937,E2 -11517.937} C_VEL
LIN {X 0,Y 390.549,Z 139.833,A -85,B 0,C 180,E1 -11520,E2 -11520} C_VEL
LIN {X 0,Y 390.313,Z 139.868,A -85,B 0,C 180,E1 -11523.097,E2 -11523.097} C_VEL
LIN {X 0,Y 390.323,Z 139.861,A -85,B 0,C 180,E1 -11526.202,E2 -11526.202} C_VEL
LIN {X 0,Y 390.204,Z 139.878,A -85,B 0,C 180,E1 -11529.329,E2 -11529.329} C_VEL
LIN {X 0,Y 390.193,Z 139.878,A -85,B 0,C 180,E1 -11533.439,E2 -11533.439} C_VEL
LIN {X 0,Y 390.148,Z 139.884,A -85,B 0,C 180,E1 -11537.308,E2 -11537.308} C_VEL
LIN {X 0,Y 390.087,Z 139.896,A -85,B 0,C 180,E1 -11540.47,E2 -11540.47} C_VEL
LIN {X 0,Y 390.078,Z 139.898,A -85,B 0,C 180,E1 -11544.481,E2 -11544.481} C_VEL
LIN {X 0,Y 390.117,Z 139.889,A -85,B 0,C 180,E1 -11547.93,E2 -11547.93} C_VEL
LIN {X 0,Y 390.023,Z 139.899,A -85,B 0,C 180,E1 -11551.505,E2 -11551.505} C_VEL
LIN {X 0,Y 390.085,Z 139.891,A -85,B 0,C 180,E1 -11555.207,E2 -11555.207} C_VEL
LIN {X 0,Y 390.095,Z 139.889,A -85,B 0,C 180,E1 -11559.092,E2 -11559.092} C_VEL
LIN {X 0,Y 390.081,Z 139.894,A -85,B 0,C 180,E1 -11562.381,E2 -11562.381} C_VEL
LIN {X 0,Y 390.056,Z 139.899,A -85,B 0,C 180,E1 -11566.114,E2 -11566.114} C_VEL
LIN {X 0,Y 390.076,Z 139.895,A -85,B 0,C 180,E1 -11569.563,E2 -11569.563} C_VEL
LIN {X 0,Y 390.048,Z 139.896,A -85,B 0,C 180,E1 -11572.449,E2 -11572.449} C_VEL
LIN {X 0,Y 390.086,Z 139.896,A -85,B 0,C 180,E1 -11576.047,E2 -11576.047} C_VEL
LIN {X 0,Y 390.048,Z 139.9,A -85,B 0,C 180,E1 -11579.869,E2 -11579.869} C_VEL
LIN {X 0,Y 390.122,Z 140.028,A -85,B 0,C 180,E1 -11580.452,E2 -11580.452} C_VEL
LIN {X 0,Y 392.692,Z 152.185,A -85,B 0,C 180,E1 -11583.135,E2 -11583.135} C_VEL
LIN {X 0,Y 393.67,Z 157.849,A -85,B 0,C 180,E1 -11584.347,E2 -11584.347} C_VEL
LIN {X 0,Y 392.425,Z 174.463,A -85,B 0,C 180,E1 -11587.631,E2 -11587.631} C_VEL
LIN {X 0,Y 391.757,Z 185.426,A -85,B 0,C 180,E1 -11589.78,E2 -11589.78} C_VEL
LIN {X 0,Y 396.185,Z 218.299,A -85,B 0,C 180,E1 -11590.648,E2 -11590.648} C_VEL
LIN {X 0,Y 395.026,Z 294.938,A -85,B 0,C 180,E1 -11592.128,E2 -11592.128} C_VEL
LIN {X 0,Y 394.424,Z 308.583,A -85,B 0,C 180,E1 -11592.602,E2 -11592.602} C_VEL
LIN {X 0,Y 393.65,Z 321.459,A -85,B 0,C 180,E1 -11593.269,E2 -11593.269} C_VEL
LIN {X 0,Y 392.717,Z 334.03,A -85,B 0,C 180,E1 -11594.162,E2 -11594.162} C_VEL
LIN {X 0,Y 391.875,Z 345.276,A -85,B 0,C 180,E1 -11595.193,E2 -11595.193} C_VEL
LIN {X 0,Y 390.989,Z 356.38,A -85,B 0,C 180,E1 -11596.487,E2 -11596.487} C_VEL
LIN {X 0,Y 390.324,Z 365.381,A -85,B 0,C 180,E1 -11597.786,E2 -11597.786} C_VEL
LIN {X 0,Y 389.567,Z 374.151,A -85,B 0,C 180,E1 -11599.344,E2 -11599.344} C_VEL
LIN {X 0,Y 389.146,Z 381.147,A -85,B 0,C 180,E1 -11600.908,E2 -11600.908} C_VEL
LIN {X 0,Y 388.895,Z 387.567,A -85,B 0,C 180,E1 -11602.733,E2 -11602.733} C_VEL
LIN {X 0,Y 388.734,Z 391.624,A -85,B 0,C 180,E1 -11604.24,E2 -11604.24} C_VEL
LIN {X 0,Y 388.736,Z 394.858,A -85,B 0,C 180,E1 -11605.853,E2 -11605.853} C_VEL
LIN {X 0,Y 388.759,Z 396.391,A -85,B 0,C 180,E1 -11606.891,E2 -11606.891} C_VEL
LIN {X 0,Y 388.842,Z 397.462,A -85,B 0,C 180,E1 -11607.928,E2 -11607.928} C_VEL
LIN {X 0,Y 388.806,Z 398.119,A -85,B 0,C 180,E1 -11608.964,E2 -11608.964} C_VEL
LIN {X 0,Y 388.8,Z 398.382,A -85,B 0,C 180,E1 -11610,E2 -11610} C_VEL
LIN {X 0,Y 388.795,Z 398.242,A -85,B 0,C 180,E1 -11611.036,E2 -11611.036} C_VEL
LIN {X 0,Y 388.814,Z 397.66,A -85,B 0,C 180,E1 -11612.072,E2 -11612.072} C_VEL
LIN {X 0,Y 388.731,Z 395.281,A -85,B 0,C 180,E1 -11614.147,E2 -11614.147} C_VEL
LIN {X 0,Y 388.747,Z 393.464,A -85,B 0,C 180,E1 -11615.186,E2 -11615.186} C_VEL
LIN {X 0,Y 388.818,Z 389.861,A -85,B 0,C 180,E1 -11616.747,E2 -11616.747} C_VEL
LIN {X 0,Y 389.026,Z 385.15,A -85,B 0,C 180,E1 -11618.31,E2 -11618.31} C_VEL
LIN {X 0,Y 389.475,Z 378.045,A -85,B 0,C 180,E1 -11620.133,E2 -11620.133} C_VEL
LIN {X 0,Y 390.128,Z 370.381,A -85,B 0,C 180,E1 -11621.693,E2 -11621.693} C_VEL
LIN {X 0,Y 390.823,Z 362.577,A -85,B 0,C 180,E1 -11622.99,E2 -11622.99} C_VEL
LIN {X 0,Y 391.612,Z 353.149,A -85,B 0,C 180,E1 -11624.279,E2 -11624.279} C_VEL
LIN {X 0,Y 392.55,Z 342.603,A -85,B 0,C 180,E1 -11625.445,E2 -11625.445} C_VEL
LIN {X 0,Y 393.615,Z 330.996,A -85,B 0,C 180,E1 -11626.466,E2 -11626.466} C_VEL
LIN {X 0,Y 394.525,Z 318.789,A -85,B 0,C 180,E1 -11627.293,E2 -11627.293} C_VEL
LIN {X 0,Y 395.417,Z 305.306,A -85,B 0,C 180,E1 -11627.954,E2 -11627.954} C_VEL
LIN {X 0,Y 396.076,Z 292.909,A -85,B 0,C 180,E1 -11628.358,E2 -11628.358} C_VEL
LIN {X 0,Y 397.158,Z 216.945,A -85,B 0,C 180,E1 -11629.844,E2 -11629.844} C_VEL
LIN {X 0,Y 394.319,Z 196.841,A -85,B 0,C 180,E1 -11630.418,E2 -11630.418} C_VEL
LIN {X 0,Y 392.073,Z 183.779,A -85,B 0,C 180,E1 -11630.83,E2 -11630.83} C_VEL
LIN {X 0,Y 393.645,Z 163.503,A -85,B 0,C 180,E1 -11634.806,E2 -11634.806} C_VEL
LIN {X 0,Y 393.934,Z 157.951,A -85,B 0,C 180,E1 -11635.918,E2 -11635.918} C_VEL
LIN {X 0,Y 391.679,Z 146.497,A -85,B 0,C 180,E1 -11638.451,E2 -11638.451} C_VEL
LIN {X 0,Y 390.06,Z 139.9,A -85,B 0,C 180,E1 -11640.034,E2 -11640.034} C_VEL
LIN {X 0,Y 390.069,Z 139.9,A -85,B 0,C 180,E1 -11643.954,E2 -11643.954} C_VEL
LIN {X 0,Y 390.048,Z 139.902,A -85,B 0,C 180,E1 -11647.551,E2 -11647.551} C_VEL
LIN {X 0,Y 390.078,Z 139.897,A -85,B 0,C 180,E1 -11650.825,E2 -11650.825} C_VEL
LIN {X 0,Y 390.056,Z 139.901,A -85,B 0,C 180,E1 -11653.886,E2 -11653.886} C_VEL
LIN {X 0,Y 390.08,Z 139.898,A -85,B 0,C 180,E1 -11657.619,E2 -11657.619} C_VEL
LIN {X 0,Y 390.094,Z 139.889,A -85,B 0,C 180,E1 -11660.908,E2 -11660.908} C_VEL
LIN {X 0,Y 390.085,Z 139.891,A -85,B 0,C 180,E1 -11664.793,E2 -11664.793} C_VEL
LIN {X 0,Y 390.023,Z 139.901,A -85,B 0,C 180,E1 -11668.495,E2 -11668.495} C_VEL
LIN {X 0,Y 390.116,Z 139.89,A -85,B 0,C 180,E1 -11672.07,E2 -11672.07} C_VEL
LIN {X 0,Y 390.076,Z 139.895,A -85,B 0,C 180,E1 -11675.519,E2 -11675.519} C_VEL
LIN {X 0,Y 390.086,Z 139.894,A -85,B 0,C 180,E1 -11679.53,E2 -11679.53} C_VEL
LIN {X 0,Y 390.137,Z 139.888,A -85,B 0,C 180,E1 -11683.248,E2 -11683.248} C_VEL
LIN {X 0,Y 390.193,Z 139.878,A -85,B 0,C 180,E1 -11686.561,E2 -11686.561} C_VEL
LIN {X 0,Y 390.203,Z 139.878,A -85,B 0,C 180,E1 -11690.671,E2 -11690.671} C_VEL
LIN {X 0,Y 390.317,Z 139.86,A -85,B 0,C 180,E1 -11692.759,E2 -11692.759} C_VEL
LIN {X 0,Y 390.225,Z 139.878,A -85,B 0,C 180,E1 -11694.833,E2 -11694.833} C_VEL
LIN {X 0,Y 390.418,Z 139.851,A -85,B 0,C 180,E1 -11697.937,E2 -11697.937} C_VEL
LIN {X 0,Y 390.548,Z 139.831,A -85,B 0,C 180,E1 -11700,E2 -11700} C_VEL
LIN {X 0,Y 390.313,Z 139.864,A -85,B 0,C 180,E1 -11703.096,E2 -11703.096} C_VEL
LIN {X 0,Y 390.3,Z 139.863,A -85,B 0,C 180,E1 -11706.561,E2 -11706.561} C_VEL
LIN {X 0,Y 390.203,Z 139.88,A -85,B 0,C 180,E1 -11709.329,E2 -11709.329} C_VEL
LIN {X 0,Y 390.192,Z 139.879,A -85,B 0,C 180,E1 -11713.438,E2 -11713.438} C_VEL
LIN {X 0,Y 390.146,Z 139.886,A -85,B 0,C 180,E1 -11717.308,E2 -11717.308} C_VEL
LIN {X 0,Y 390.085,Z 139.897,A -85,B 0,C 180,E1 -11720.47,E2 -11720.47} C_VEL
LIN {X 0,Y 390.087,Z 139.898,A -85,B 0,C 180,E1 -11723.351,E2 -11723.351} C_VEL
LIN {X 0,Y 390.111,Z 139.894,A -85,B 0,C 180,E1 -11726.768,E2 -11726.768} C_VEL
LIN {X 0,Y 390.09,Z 139.92,A -85,B 0,C 180,E1 -11730.52,E2 -11730.52} C_VEL
LIN {X 0,Y 391.48,Z 146.301,A -85,B 0,C 180,E1 -11732.184,E2 -11732.184} C_VEL
LIN {X 0,Y 396.547,Z 159.758,A -85,B 0,C 180,E1 -11732.796,E2 -11732.796} C_VEL
LIN {X 0,Y 398.066,Z 166.808,A -85,B 0,C 180,E1 -11733.032,E2 -11733.032} C_VEL
LIN {X 0,Y 396.474,Z 254.002,A -85,B 0,C 180,E1 -11734.737,E2 -11734.737} C_VEL
LIN {X 0,Y 396.027,Z 266.772,A -85,B 0,C 180,E1 -11735.187,E2 -11735.187} C_VEL
LIN {X 0,Y 395.51,Z 278.72,A -85,B 0,C 180,E1 -11735.804,E2 -11735.804} C_VEL
LIN {X 0,Y 394.774,Z 290.684,A -85,B 0,C 180,E1 -11736.633,E2 -11736.633} C_VEL
LIN {X 0,Y 393.946,Z 301.917,A -85,B 0,C 180,E1 -11737.643,E2 -11737.643} C_VEL
LIN {X 0,Y 393.104,Z 311.708,A -85,B 0,C 180,E1 -11738.736,E2 -11738.736} C_VEL
LIN {X 0,Y 392.254,Z 320.688,A -85,B 0,C 180,E1 -11739.963,E2 -11739.963} C_VEL
LIN {X 0,Y 391.376,Z 329.303,A -85,B 0,C 180,E1 -11741.412,E2 -11741.412} C_VEL
LIN {X 0,Y 390.586,Z 336.293,A -85,B 0,C 180,E1 -11742.863,E2 -11742.863} C_VEL
LIN {X 0,Y 389.962,Z 343.137,A -85,B 0,C 180,E1 -11744.657,E2 -11744.657} C_VEL
LIN {X 0,Y 389.535,Z 347.673,A -85,B 0,C 180,E1 -11746.193,E2 -11746.193} C_VEL
LIN {X 0,Y 389.127,Z 351.772,A -85,B 0,C 180,E1 -11748.068,E2 -11748.068} C_VEL
LIN {X 0,Y 388.902,Z 353.825,A -85,B 0,C 180,E1 -11749.416,E2 -11749.416} C_VEL
LIN {X 0,Y 388.745,Z 355.346,A -85,B 0,C 180,E1 -11751.021,E2 -11751.021} C_VEL
LIN {X 0,Y 388.708,Z 355.911,A -85,B 0,C 180,E1 -11752.706,E2 -11752.706} C_VEL
LIN {X 0,Y 388.73,Z 355.251,A -85,B 0,C 180,E1 -11754.652,E2 -11754.652} C_VEL
LIN {X 0,Y 388.814,Z 353.656,A -85,B 0,C 180,E1 -11756.25,E2 -11756.25} C_VEL
LIN {X 0,Y 389.094,Z 350.547,A -85,B 0,C 180,E1 -11758.096,E2 -11758.096} C_VEL
LIN {X 0,Y 389.465,Z 345.825,A -85,B 0,C 180,E1 -11760.017,E2 -11760.017} C_VEL
LIN {X 0,Y 389.88,Z 340.008,A -85,B 0,C 180,E1 -11761.76,E2 -11761.76} C_VEL
LIN {X 0,Y 390.535,Z 332.581,A -85,B 0,C 180,E1 -11763.482,E2 -11763.482} C_VEL
LIN {X 0,Y 391.229,Z 324.203,A -85,B 0,C 180,E1 -11765.03,E2 -11765.03} C_VEL
LIN {X 0,Y 391.999,Z 315.157,A -85,B 0,C 180,E1 -11766.37,E2 -11766.37} C_VEL
LIN {X 0,Y 392.804,Z 304.448,A -85,B 0,C 180,E1 -11767.654,E2 -11767.654} C_VEL
LIN {X 0,Y 393.655,Z 293.055,A -85,B 0,C 180,E1 -11768.735,E2 -11768.735} C_VEL
LIN {X 0,Y 394.36,Z 280.384,A -85,B 0,C 180,E1 -11769.665,E2 -11769.665} C_VEL
LIN {X 0,Y 394.935,Z 268.036,A -85,B 0,C 180,E1 -11770.34,E2 -11770.34} C_VEL
LIN {X 0,Y 395.292,Z 256.104,A -85,B 0,C 180,E1 -11770.796,E2 -11770.796} C_VEL
LIN {X 0,Y 395.591,Z 240.431,A -85,B 0,C 180,E1 -11771.152,E2 -11771.152} C_VEL
LIN {X 0,Y 396.593,Z 165.279,A -85,B 0,C 180,E1 -11772.584,E2 -11772.584} C_VEL
LIN {X 0,Y 393.738,Z 152.734,A -85,B 0,C 180,E1 -11772.972,E2 -11772.972} C_VEL
LIN {X 0,Y 391.127,Z 144.877,A -85,B 0,C 180,E1 -11773.292,E2 -11773.292} C_VEL
LIN {X 0,Y 390.177,Z 139.883,A -85,B 0,C 180,E1 -11774.593,E2 -11774.593} C_VEL
LIN {X 0,Y 390.166,Z 139.887,A -85,B 0,C 180,E1 -11777.517,E2 -11777.517} C_VEL
LIN {X 0,Y 390.165,Z 139.883,A -85,B 0,C 180,E1 -11779.977,E2 -11779.977} C_VEL
LIN {X 0,Y 389.526,Z 139.962,A -85,B 0,C 180,E1 -11780.84,E2 -11780.84} C_VEL
LIN {X 0,Y 386.724,Z 140.31,A -85,B 0,C 180,E1 -11782.243,E2 -11782.243} C_VEL
LIN {X 0,Y 384.332,Z 140.612,A -85,B 0,C 180,E1 -11783.376,E2 -11783.376} C_VEL
LIN {X 0,Y 383.293,Z 140.737,A -85,B 0,C 180,E1 -11784.252,E2 -11784.252} C_VEL
LIN {X 0,Y 383.202,Z 140.748,A -85,B 0,C 180,E1 -11784.549,E2 -11784.549} C_VEL
LIN {X 0,Y 383.385,Z 140.727,A -85,B 0,C 180,E1 -11787.899,E2 -11787.899} C_VEL
LIN {X 0,Y 383.518,Z 140.71,A -85,B 0,C 180,E1 -11790,E2 -11790} C_VEL
LIN {X 0,Y 383.246,Z 140.748,A -85,B 0,C 180,E1 -11793.154,E2 -11793.154} C_VEL
LIN {X 0,Y 383.256,Z 140.741,A -85,B 0,C 180,E1 -11796.317,E2 -11796.317} C_VEL
LIN {X 0,Y 383.143,Z 140.758,A -85,B 0,C 180,E1 -11799.502,E2 -11799.502} C_VEL
LIN {X 0,Y 383.125,Z 140.759,A -85,B 0,C 180,E1 -11803.536,E2 -11803.536} C_VEL
LIN {X 0,Y 383.093,Z 140.767,A -85,B 0,C 180,E1 -11807.069,E2 -11807.069} C_VEL
LIN {X 0,Y 383.028,Z 140.774,A -85,B 0,C 180,E1 -11810.647,E2 -11810.647} C_VEL
LIN {X 0,Y 383.025,Z 140.77,A -85,B 0,C 180,E1 -11813.808,E2 -11813.808} C_VEL
LIN {X 0,Y 383.079,Z 140.765,A -85,B 0,C 180,E1 -11816.123,E2 -11816.123} C_VEL
LIN {X 0,Y 383.04,Z 140.773,A -85,B 0,C 180,E1 -11818.493,E2 -11818.493} C_VEL
LIN {X 0,Y 383.008,Z 140.775,A -85,B 0,C 180,E1 -11822.15,E2 -11822.15} C_VEL
LIN {X 0,Y 383.016,Z 140.776,A -85,B 0,C 180,E1 -11824.668,E2 -11824.668} C_VEL
LIN {X 0,Y 382.997,Z 140.775,A -85,B 0,C 180,E1 -11827.903,E2 -11827.903} C_VEL
LIN {X 0,Y 382.982,Z 140.775,A -85,B 0,C 180,E1 -11831.347,E2 -11831.347} C_VEL
LIN {X 0,Y 382.995,Z 140.78,A -85,B 0,C 180,E1 -11834.303,E2 -11834.303} C_VEL
LIN {X 0,Y 383.008,Z 140.772,A -85,B 0,C 180,E1 -11837.24,E2 -11837.24} C_VEL
LIN {X 0,Y 383.015,Z 140.774,A -85,B 0,C 180,E1 -11840.413,E2 -11840.413} C_VEL
LIN {X 0,Y 383.025,Z 140.776,A -85,B 0,C 180,E1 -11844.045,E2 -11844.045} C_VEL
LIN {X 0,Y 382.985,Z 140.778,A -85,B 0,C 180,E1 -11847.578,E2 -11847.578} C_VEL
LIN {X 0,Y 382.99,Z 140.776,A -85,B 0,C 180,E1 -11850.3,E2 -11850.3} C_VEL
LIN {X 0,Y 383.055,Z 140.766,A -85,B 0,C 180,E1 -11852.698,E2 -11852.698} C_VEL
LIN {X 0,Y 383.049,Z 140.768,A -85,B 0,C 180,E1 -11855.04,E2 -11855.04} C_VEL
LIN {X 0,Y 382.993,Z 140.774,A -85,B 0,C 180,E1 -11858.469,E2 -11858.469} C_VEL
LIN {X 0,Y 383.087,Z 140.766,A -85,B 0,C 180,E1 -11861.828,E2 -11861.828} C_VEL
LIN {X 0,Y 383.109,Z 140.763,A -85,B 0,C 180,E1 -11865.118,E2 -11865.118} C_VEL
LIN {X 0,Y 383.096,Z 140.761,A -85,B 0,C 180,E1 -11868.358,E2 -11868.358} C_VEL
LIN {X 0,Y 383.302,Z 140.736,A -85,B 0,C 180,E1 -11871.933,E2 -11871.933} C_VEL
LIN {X 0,Y 383.198,Z 140.75,A -85,B 0,C 180,E1 -11874.739,E2 -11874.739} C_VEL
LIN {X 0,Y 383.386,Z 140.726,A -85,B 0,C 180,E1 -11877.899,E2 -11877.899} C_VEL
LIN {X 0,Y 383.518,Z 140.709,A -85,B 0,C 180,E1 -11880,E2 -11880} C_VEL
LIN {X 0,Y 383.249,Z 140.747,A -85,B 0,C 180,E1 -11883.154,E2 -11883.154} C_VEL
LIN {X 0,Y 383.279,Z 140.739,A -85,B 0,C 180,E1 -11886.317,E2 -11886.317} C_VEL
LIN {X 0,Y 383.15,Z 140.755,A -85,B 0,C 180,E1 -11889.502,E2 -11889.502} C_VEL
LIN {X 0,Y 383.124,Z 140.758,A -85,B 0,C 180,E1 -11893.536,E2 -11893.536} C_VEL
LIN {X 0,Y 383.094,Z 140.762,A -85,B 0,C 180,E1 -11897.455,E2 -11897.455} C_VEL
LIN {X 0,Y 383.028,Z 140.776,A -85,B 0,C 180,E1 -11900.647,E2 -11900.647} C_VEL
LIN {X 0,Y 383.025,Z 140.771,A -85,B 0,C 180,E1 -11903.808,E2 -11903.808} C_VEL
LIN {X 0,Y 383.079,Z 140.766,A -85,B 0,C 180,E1 -11906.124,E2 -11906.124} C_VEL
LIN {X 0,Y 383.04,Z 140.774,A -85,B 0,C 180,E1 -11908.493,E2 -11908.493} C_VEL
LIN {X 0,Y 383.009,Z 140.777,A -85,B 0,C 180,E1 -11912.15,E2 -11912.15} C_VEL
LIN {X 0,Y 383.018,Z 140.773,A -85,B 0,C 180,E1 -11914.668,E2 -11914.668} C_VEL
LIN {X 0,Y 383.003,Z 140.777,A -85,B 0,C 180,E1 -11917.905,E2 -11917.905} C_VEL
LIN {X 0,Y 383.014,Z 140.772,A -85,B 0,C 180,E1 -11921.344,E2 -11921.344} C_VEL
LIN {X 0,Y 382.997,Z 140.777,A -85,B 0,C 180,E1 -11924.304,E2 -11924.304} C_VEL
LIN {X 0,Y 383.04,Z 140.769,A -85,B 0,C 180,E1 -11927.245,E2 -11927.245} C_VEL
LIN {X 0,Y 383.022,Z 140.772,A -85,B 0,C 180,E1 -11930.413,E2 -11930.413} C_VEL
LIN {X 0,Y 383.028,Z 140.773,A -85,B 0,C 180,E1 -11934.045,E2 -11934.045} C_VEL
LIN {X 0,Y 382.988,Z 140.78,A -85,B 0,C 180,E1 -11937.578,E2 -11937.578} C_VEL
LIN {X 0,Y 383.05,Z 140.845,A -85,B 0,C 180,E1 -11940.158,E2 -11940.158} C_VEL
LIN {X 0,Y 385.898,Z 154.259,A -85,B 0,C 180,E1 -11943.176,E2 -11943.176} C_VEL
LIN {X 0,Y 386.712,Z 160.079,A -85,B 0,C 180,E1 -11944.429,E2 -11944.429} C_VEL
LIN {X 0,Y 385.253,Z 178.337,A -85,B 0,C 180,E1 -11948.096,E2 -11948.096} C_VEL
LIN {X 0,Y 384.843,Z 184.964,A -85,B 0,C 180,E1 -11949.418,E2 -11949.418} C_VEL
LIN {X 0,Y 389.402,Z 218.835,A -85,B 0,C 180,E1 -11950.349,E2 -11950.349} C_VEL
LIN {X 0,Y 388.228,Z 294.5,A -85,B 0,C 180,E1 -11951.838,E2 -11951.838} C_VEL
LIN {X 0,Y 387.603,Z 308.156,A -85,B 0,C 180,E1 -11952.319,E2 -11952.319} C_VEL
LIN {X 0,Y 386.827,Z 320.535,A -85,B 0,C 180,E1 -11952.965,E2 -11952.965} C_VEL
LIN {X 0,Y 386.021,Z 331.641,A -85,B 0,C 180,E1 -11953.745,E2 -11953.745} C_VEL
LIN {X 0,Y 385.042,Z 343.243,A -85,B 0,C 180,E1 -11954.789,E2 -11954.789} C_VEL
LIN {X 0,Y 384.244,Z 353.522,A -85,B 0,C 180,E1 -11955.95,E2 -11955.95} C_VEL
LIN {X 0,Y 383.412,Z 363.129,A -85,B 0,C 180,E1 -11957.293,E2 -11957.293} C_VEL
LIN {X 0,Y 382.78,Z 370.866,A -85,B 0,C 180,E1 -11958.617,E2 -11958.617} C_VEL
LIN {X 0,Y 382.242,Z 378.444,A -85,B 0,C 180,E1 -11960.208,E2 -11960.208} C_VEL
LIN {X 0,Y 381.88,Z 385.436,A -85,B 0,C 180,E1 -11962.066,E2 -11962.066} C_VEL
LIN {X 0,Y 381.674,Z 390.61,A -85,B 0,C 180,E1 -11963.901,E2 -11963.901} C_VEL
LIN {X 0,Y 381.66,Z 394.417,A -85,B 0,C 180,E1 -11965.776,E2 -11965.776} C_VEL
LIN {X 0,Y 381.662,Z 395.963,A -85,B 0,C 180,E1 -11966.833,E2 -11966.833} C_VEL
LIN {X 0,Y 381.755,Z 397.051,A -85,B 0,C 180,E1 -11967.89,E2 -11967.89} C_VEL
LIN {X 0,Y 381.736,Z 397.718,A -85,B 0,C 180,E1 -11968.945,E2 -11968.945} C_VEL
LIN {X 0,Y 381.726,Z 397.988,A -85,B 0,C 180,E1 -11970,E2 -11970} C_VEL
LIN {X 0,Y 381.725,Z 397.86,A -85,B 0,C 180,E1 -11971.055,E2 -11971.055} C_VEL
LIN {X 0,Y 381.728,Z 397.29,A -85,B 0,C 180,E1 -11972.11,E2 -11972.11} C_VEL
LIN {X 0,Y 381.653,Z 394.924,A -85,B 0,C 180,E1 -11974.224,E2 -11974.224} C_VEL
LIN {X 0,Y 381.634,Z 391.535,A -85,B 0,C 180,E1 -11976.042,E2 -11976.042} C_VEL
LIN {X 0,Y 381.882,Z 386.506,A -85,B 0,C 180,E1 -11977.934,E2 -11977.934} C_VEL
LIN {X 0,Y 382.256,Z 379.966,A -85,B 0,C 180,E1 -11979.792,E2 -11979.792} C_VEL
LIN {X 0,Y 382.833,Z 372.872,A -85,B 0,C 180,E1 -11981.382,E2 -11981.382} C_VEL
LIN {X 0,Y 383.746,Z 364.012,A -85,B 0,C 180,E1 -11982.964,E2 -11982.964} C_VEL
LIN {X 0,Y 384.626,Z 353.839,A -85,B 0,C 180,E1 -11984.434,E2 -11984.434} C_VEL
LIN {X 0,Y 385.591,Z 343.809,A -85,B 0,C 180,E1 -11985.595,E2 -11985.595} C_VEL
LIN {X 0,Y 386.667,Z 332.556,A -85,B 0,C 180,E1 -11986.635,E2 -11986.635} C_VEL
LIN {X 0,Y 387.683,Z 319.98,A -85,B 0,C 180,E1 -11987.54,E2 -11987.54} C_VEL
LIN {X 0,Y 388.614,Z 307.131,A -85,B 0,C 180,E1 -11988.211,E2 -11988.211} C_VEL
LIN {X 0,Y 389.339,Z 293.602,A -85,B 0,C 180,E1 -11988.687,E2 -11988.687} C_VEL
LIN {X 0,Y 390.577,Z 217.945,A -85,B 0,C 180,E1 -11990.202,E2 -11990.202} C_VEL
LIN {X 0,Y 387.352,Z 195.265,A -85,B 0,C 180,E1 -11990.873,E2 -11990.873} C_VEL
LIN {X 0,Y 385.23,Z 183.34,A -85,B 0,C 180,E1 -11991.267,E2 -11991.267} C_VEL
LIN {X 0,Y 386.773,Z 164.701,A -85,B 0,C 180,E1 -11994.991,E2 -11994.991} C_VEL
LIN {X 0,Y 387.022,Z 159.177,A -85,B 0,C 180,E1 -11996.121,E2 -11996.121} C_VEL
LIN {X 0,Y 385.12,Z 149.421,A -85,B 0,C 180,E1 -11998.325,E2 -11998.325} C_VEL
LIN {X 0,Y 382.999,Z 140.78,A -85,B 0,C 180,E1 -12000.407,E2 -12000.407} C_VEL
LIN {X 0,Y 383.004,Z 140.778,A -85,B 0,C 180,E1 -12003.4,E2 -12003.4} C_VEL
LIN {X 0,Y 383.035,Z 140.779,A -85,B 0,C 180,E1 -12006.165,E2 -12006.165} C_VEL
LIN {X 0,Y 383.02,Z 140.781,A -85,B 0,C 180,E1 -12009.957,E2 -12009.957} C_VEL
LIN {X 0,Y 383.033,Z 140.775,A -85,B 0,C 180,E1 -12012.783,E2 -12012.783} C_VEL
LIN {X 0,Y 382.998,Z 140.779,A -85,B 0,C 180,E1 -12015.789,E2 -12015.789} C_VEL
LIN {X 0,Y 383.015,Z 140.774,A -85,B 0,C 180,E1 -12018.791,E2 -12018.791} C_VEL
LIN {X 0,Y 383.003,Z 140.779,A -85,B 0,C 180,E1 -12022.095,E2 -12022.095} C_VEL
LIN {X 0,Y 383.018,Z 140.774,A -85,B 0,C 180,E1 -12025.332,E2 -12025.332} C_VEL
LIN {X 0,Y 382.982,Z 140.778,A -85,B 0,C 180,E1 -12029.081,E2 -12029.081} C_VEL
LIN {X 0,Y 383.055,Z 140.767,A -85,B 0,C 180,E1 -12032.698,E2 -12032.698} C_VEL
LIN {X 0,Y 383.049,Z 140.766,A -85,B 0,C 180,E1 -12035.039,E2 -12035.039} C_VEL
LIN {X 0,Y 382.991,Z 140.773,A -85,B 0,C 180,E1 -12038.469,E2 -12038.469} C_VEL
LIN {X 0,Y 383.088,Z 140.763,A -85,B 0,C 180,E1 -12041.827,E2 -12041.827} C_VEL
LIN {X 0,Y 383.109,Z 140.757,A -85,B 0,C 180,E1 -12045.118,E2 -12045.118} C_VEL
LIN {X 0,Y 383.096,Z 140.758,A -85,B 0,C 180,E1 -12048.358,E2 -12048.358} C_VEL
LIN {X 0,Y 383.302,Z 140.733,A -85,B 0,C 180,E1 -12051.933,E2 -12051.933} C_VEL
LIN {X 0,Y 383.198,Z 140.752,A -85,B 0,C 180,E1 -12054.738,E2 -12054.738} C_VEL
LIN {X 0,Y 383.386,Z 140.727,A -85,B 0,C 180,E1 -12057.899,E2 -12057.899} C_VEL
LIN {X 0,Y 383.518,Z 140.707,A -85,B 0,C 180,E1 -12060,E2 -12060} C_VEL
LIN {X 0,Y 383.249,Z 140.744,A -85,B 0,C 180,E1 -12063.153,E2 -12063.153} C_VEL
LIN {X 0,Y 383.261,Z 140.74,A -85,B 0,C 180,E1 -12066.551,E2 -12066.551} C_VEL
LIN {X 0,Y 383.149,Z 140.758,A -85,B 0,C 180,E1 -12069.502,E2 -12069.502} C_VEL
LIN {X 0,Y 383.123,Z 140.76,A -85,B 0,C 180,E1 -12073.536,E2 -12073.536} C_VEL
LIN {X 0,Y 383.092,Z 140.764,A -85,B 0,C 180,E1 -12077.455,E2 -12077.455} C_VEL
LIN {X 0,Y 383.027,Z 140.778,A -85,B 0,C 180,E1 -12080.647,E2 -12080.647} C_VEL
LIN {X 0,Y 383.031,Z 140.778,A -85,B 0,C 180,E1 -12083.807,E2 -12083.807} C_VEL
LIN {X 0,Y 383.077,Z 140.769,A -85,B 0,C 180,E1 -12086.123,E2 -12086.123} C_VEL
LIN {X 0,Y 383.065,Z 140.769,A -85,B 0,C 180,E1 -12090.127,E2 -12090.127} C_VEL
LIN {X 0,Y 384.409,Z 146.934,A -85,B 0,C 180,E1 -12091.749,E2 -12091.749} C_VEL
LIN {X 0,Y 390.241,Z 161.912,A -85,B 0,C 180,E1 -12092.449,E2 -12092.449} C_VEL
LIN {X 0,Y 391.495,Z 168.198,A -85,B 0,C 180,E1 -12092.661,E2 -12092.661} C_VEL
LIN {X 0,Y 389.822,Z 254.585,A -85,B 0,C 180,E1 -12094.386,E2 -12094.386} C_VEL
LIN {X 0,Y 389.355,Z 267.383,A -85,B 0,C 180,E1 -12094.848,E2 -12094.848} C_VEL
LIN {X 0,Y 388.777,Z 279.771,A -85,B 0,C 180,E1 -12095.504,E2 -12095.504} C_VEL
LIN {X 0,Y 388.087,Z 290.386,A -85,B 0,C 180,E1 -12096.25,E2 -12096.25} C_VEL
LIN {X 0,Y 387.245,Z 301.488,A -85,B 0,C 180,E1 -12097.249,E2 -12097.249} C_VEL
LIN {X 0,Y 386.234,Z 312.68,A -85,B 0,C 180,E1 -12098.516,E2 -12098.516} C_VEL
LIN {X 0,Y 385.353,Z 321.536,A -85,B 0,C 180,E1 -12099.76,E2 -12099.76} C_VEL
LIN {X 0,Y 384.476,Z 329.627,A -85,B 0,C 180,E1 -12101.152,E2 -12101.152} C_VEL
LIN {X 0,Y 383.528,Z 337.615,A -85,B 0,C 180,E1 -12102.863,E2 -12102.863} C_VEL
LIN {X 0,Y 382.895,Z 344.169,A -85,B 0,C 180,E1 -12104.664,E2 -12104.664} C_VEL
LIN {X 0,Y 382.406,Z 349.083,A -85,B 0,C 180,E1 -12106.453,E2 -12106.453} C_VEL
LIN {X 0,Y 381.982,Z 353.115,A -85,B 0,C 180,E1 -12108.521,E2 -12108.521} C_VEL
LIN {X 0,Y 381.676,Z 355.524,A -85,B 0,C 180,E1 -12110.657,E2 -12110.657} C_VEL
LIN {X 0,Y 381.635,Z 356.29,A -85,B 0,C 180,E1 -12112.576,E2 -12112.576} C_VEL
LIN {X 0,Y 381.603,Z 355.939,A -85,B 0,C 180,E1 -12114.13,E2 -12114.13} C_VEL
LIN {X 0,Y 381.713,Z 354.435,A -85,B 0,C 180,E1 -12115.948,E2 -12115.948} C_VEL
LIN {X 0,Y 381.968,Z 351.617,A -85,B 0,C 180,E1 -12117.819,E2 -12117.819} C_VEL
LIN {X 0,Y 382.316,Z 347.155,A -85,B 0,C 180,E1 -12119.767,E2 -12119.767} C_VEL
LIN {X 0,Y 382.749,Z 341.84,A -85,B 0,C 180,E1 -12121.484,E2 -12121.484} C_VEL
LIN {X 0,Y 383.434,Z 334.477,A -85,B 0,C 180,E1 -12123.317,E2 -12123.317} C_VEL
LIN {X 0,Y 384.084,Z 326.827,A -85,B 0,C 180,E1 -12124.822,E2 -12124.822} C_VEL
LIN {X 0,Y 384.912,Z 317.439,A -85,B 0,C 180,E1 -12126.316,E2 -12126.316} C_VEL
LIN {X 0,Y 385.657,Z 308.276,A -85,B 0,C 180,E1 -12127.5,E2 -12127.5} C_VEL
LIN {X 0,Y 386.489,Z 296.942,A -85,B 0,C 180,E1 -12128.674,E2 -12128.674} C_VEL
LIN {X 0,Y 387.203,Z 286.305,A -85,B 0,C 180,E1 -12129.55,E2 -12129.55} C_VEL
LIN {X 0,Y 387.853,Z 273.646,A -85,B 0,C 180,E1 -12130.357,E2 -12130.357} C_VEL
LIN {X 0,Y 388.346,Z 260.482,A -85,B 0,C 180,E1 -12130.946,E2 -12130.946} C_VEL
LIN {X 0,Y 388.69,Z 247.505,A -85,B 0,C 180,E1 -12131.314,E2 -12131.314} C_VEL
LIN {X 0,Y 389.909,Z 166.621,A -85,B 0,C 180,E1 -12132.88,E2 -12132.88} C_VEL
LIN {X 0,Y 387.31,Z 155.112,A -85,B 0,C 180,E1 -12133.241,E2 -12133.241} C_VEL
LIN {X 0,Y 384.068,Z 145.319,A -85,B 0,C 180,E1 -12133.626,E2 -12133.626} C_VEL
LIN {X 0,Y 383.101,Z 140.765,A -85,B 0,C 180,E1 -12134.846,E2 -12134.846} C_VEL
LIN {X 0,Y 383.126,Z 140.764,A -85,B 0,C 180,E1 -12137.284,E2 -12137.284} C_VEL
LIN {X 0,Y 383.151,Z 140.754,A -85,B 0,C 180,E1 -12140.498,E2 -12140.498} C_VEL
LIN {X 0,Y 383.28,Z 140.743,A -85,B 0,C 180,E1 -12143.684,E2 -12143.684} C_VEL
LIN {X 0,Y 383.202,Z 140.748,A -85,B 0,C 180,E1 -12144.549,E2 -12144.549} C_VEL
LIN {X 0,Y 382.51,Z 140.841,A -85,B 0,C 180,E1 -12145.427,E2 -12145.427} C_VEL
LIN {X 0,Y 379.645,Z 141.196,A -85,B 0,C 180,E1 -12146.855,E2 -12146.855} C_VEL
LIN {X 0,Y 377.288,Z 141.489,A -85,B 0,C 180,E1 -12148.009,E2 -12148.009} C_VEL
LIN {X 0,Y 376.354,Z 141.603,A -85,B 0,C 180,E1 -12148.901,E2 -12148.901} C_VEL
LIN {X 0,Y 376.319,Z 141.606,A -85,B 0,C 180,E1 -12149.203,E2 -12149.203} C_VEL
LIN {X 0,Y 376.487,Z 141.585,A -85,B 0,C 180,E1 -12150,E2 -12150} C_VEL
LIN {X 0,Y 376.184,Z 141.628,A -85,B 0,C 180,E1 -12153.213,E2 -12153.213} C_VEL
LIN {X 0,Y 376.214,Z 141.619,A -85,B 0,C 180,E1 -12156.436,E2 -12156.436} C_VEL
LIN {X 0,Y 376.113,Z 141.632,A -85,B 0,C 180,E1 -12159.682,E2 -12159.682} C_VEL
LIN {X 0,Y 376.089,Z 141.635,A -85,B 0,C 180,E1 -12163.658,E2 -12163.658} C_VEL
LIN {X 0,Y 376.032,Z 141.643,A -85,B 0,C 180,E1 -12167.4,E2 -12167.4} C_VEL
LIN {X 0,Y 375.978,Z 141.655,A -85,B 0,C 180,E1 -12170.832,E2 -12170.832} C_VEL
LIN {X 0,Y 375.989,Z 141.649,A -85,B 0,C 180,E1 -12174.282,E2 -12174.282} C_VEL
LIN {X 0,Y 376.019,Z 141.649,A -85,B 0,C 180,E1 -12176.652,E2 -12176.652} C_VEL
LIN {X 0,Y 375.969,Z 141.651,A -85,B 0,C 180,E1 -12179.079,E2 -12179.079} C_VEL
LIN {X 0,Y 375.948,Z 141.655,A -85,B 0,C 180,E1 -12182.828,E2 -12182.828} C_VEL
LIN {X 0,Y 375.956,Z 141.651,A -85,B 0,C 180,E1 -12185.415,E2 -12185.415} C_VEL
LIN {X 0,Y 375.971,Z 141.654,A -85,B 0,C 180,E1 -12188.27,E2 -12188.27} C_VEL
LIN {X 0,Y 375.933,Z 141.654,A -85,B 0,C 180,E1 -12191.601,E2 -12191.601} C_VEL
LIN {X 0,Y 375.926,Z 141.654,A -85,B 0,C 180,E1 -12195.268,E2 -12195.268} C_VEL
LIN {X 0,Y 375.933,Z 141.657,A -85,B 0,C 180,E1 -12198.399,E2 -12198.399} C_VEL
LIN {X 0,Y 375.974,Z 141.651,A -85,B 0,C 180,E1 -12201.729,E2 -12201.729} C_VEL
LIN {X 0,Y 375.978,Z 141.649,A -85,B 0,C 180,E1 -12205.333,E2 -12205.333} C_VEL
LIN {X 0,Y 375.956,Z 141.652,A -85,B 0,C 180,E1 -12208.438,E2 -12208.438} C_VEL
LIN {X 0,Y 375.994,Z 141.649,A -85,B 0,C 180,E1 -12212.141,E2 -12212.141} C_VEL
LIN {X 0,Y 376.003,Z 141.645,A -85,B 0,C 180,E1 -12214.539,E2 -12214.539} C_VEL
LIN {X 0,Y 375.956,Z 141.653,A -85,B 0,C 180,E1 -12218.046,E2 -12218.046} C_VEL
LIN {X 0,Y 376.022,Z 141.648,A -85,B 0,C 180,E1 -12221.474,E2 -12221.474} C_VEL
LIN {X 0,Y 376.057,Z 141.639,A -85,B 0,C 180,E1 -12224.833,E2 -12224.833} C_VEL
LIN {X 0,Y 376.048,Z 141.64,A -85,B 0,C 180,E1 -12228.137,E2 -12228.137} C_VEL
LIN {X 0,Y 376.256,Z 141.615,A -85,B 0,C 180,E1 -12231.877,E2 -12231.877} C_VEL
LIN {X 0,Y 376.171,Z 141.625,A -85,B 0,C 180,E1 -12234.64,E2 -12234.64} C_VEL
LIN {X 0,Y 376.352,Z 141.602,A -85,B 0,C 180,E1 -12237.86,E2 -12237.86} C_VEL
LIN {X 0,Y 376.488,Z 141.585,A -85,B 0,C 180,E1 -12240,E2 -12240} C_VEL
LIN {X 0,Y 376.187,Z 141.626,A -85,B 0,C 180,E1 -12243.213,E2 -12243.213} C_VEL
LIN {X 0,Y 376.237,Z 141.617,A -85,B 0,C 180,E1 -12246.435,E2 -12246.435} C_VEL
LIN {X 0,Y 376.118,Z 141.631,A -85,B 0,C 180,E1 -12249.682,E2 -12249.682} C_VEL
LIN {X 0,Y 376.088,Z 141.634,A -85,B 0,C 180,E1 -12253.658,E2 -12253.658} C_VEL
LIN {X 0,Y 376.043,Z 141.64,A -85,B 0,C 180,E1 -12257.608,E2 -12257.608} C_VEL
LIN {X 0,Y 375.977,Z 141.652,A -85,B 0,C 180,E1 -12260.832,E2 -12260.832} C_VEL
LIN {X 0,Y 375.989,Z 141.651,A -85,B 0,C 180,E1 -12264.282,E2 -12264.282} C_VEL
LIN {X 0,Y 376.019,Z 141.647,A -85,B 0,C 180,E1 -12266.652,E2 -12266.652} C_VEL
LIN {X 0,Y 375.97,Z 141.65,A -85,B 0,C 180,E1 -12269.079,E2 -12269.079} C_VEL
LIN {X 0,Y 375.949,Z 141.653,A -85,B 0,C 180,E1 -12272.829,E2 -12272.829} C_VEL
LIN {X 0,Y 375.958,Z 141.651,A -85,B 0,C 180,E1 -12275.416,E2 -12275.416} C_VEL
LIN {X 0,Y 375.978,Z 141.653,A -85,B 0,C 180,E1 -12278.272,E2 -12278.272} C_VEL
LIN {X 0,Y 375.961,Z 141.652,A -85,B 0,C 180,E1 -12281.606,E2 -12281.606} C_VEL
LIN {X 0,Y 375.928,Z 141.655,A -85,B 0,C 180,E1 -12285.269,E2 -12285.269} C_VEL
LIN {X 0,Y 375.961,Z 141.652,A -85,B 0,C 180,E1 -12288.395,E2 -12288.395} C_VEL
LIN {X 0,Y 375.979,Z 141.654,A -85,B 0,C 180,E1 -12291.729,E2 -12291.729} C_VEL
LIN {X 0,Y 375.981,Z 141.65,A -85,B 0,C 180,E1 -12295.333,E2 -12295.333} C_VEL
LIN {X 0,Y 375.959,Z 141.651,A -85,B 0,C 180,E1 -12298.438,E2 -12298.438} C_VEL
LIN {X 0,Y 376.017,Z 141.804,A -85,B 0,C 180,E1 -12299.886,E2 -12299.886} C_VEL
LIN {X 0,Y 378.67,Z 154.112,A -85,B 0,C 180,E1 -12302.72,E2 -12302.72} C_VEL
LIN {X 0,Y 379.755,Z 160.888,A -85,B 0,C 180,E1 -12304.221,E2 -12304.221} C_VEL
LIN {X 0,Y 378.362,Z 177.499,A -85,B 0,C 180,E1 -12307.618,E2 -12307.618} C_VEL
LIN {X 0,Y 377.944,Z 184.794,A -85,B 0,C 180,E1 -12309.093,E2 -12309.093} C_VEL
LIN {X 0,Y 382.609,Z 218.846,A -85,B 0,C 180,E1 -12310.029,E2 -12310.029} C_VEL
LIN {X 0,Y 381.447,Z 293.993,A -85,B 0,C 180,E1 -12311.538,E2 -12311.538} C_VEL
LIN {X 0,Y 380.784,Z 307.684,A -85,B 0,C 180,E1 -12312.027,E2 -12312.027} C_VEL
LIN {X 0,Y 380.014,Z 319.542,A -85,B 0,C 180,E1 -12312.65,E2 -12312.65} C_VEL
LIN {X 0,Y 379.147,Z 330.819,A -85,B 0,C 180,E1 -12313.441,E2 -12313.441} C_VEL
LIN {X 0,Y 378.126,Z 342.506,A -85,B 0,C 180,E1 -12314.504,E2 -12314.504} C_VEL
LIN {X 0,Y 377.336,Z 352.054,A -85,B 0,C 180,E1 -12315.586,E2 -12315.586} C_VEL
LIN {X 0,Y 376.584,Z 360.761,A -85,B 0,C 180,E1 -12316.784,E2 -12316.784} C_VEL
LIN {X 0,Y 375.906,Z 368.857,A -85,B 0,C 180,E1 -12318.132,E2 -12318.132} C_VEL
LIN {X 0,Y 375.255,Z 376.78,A -85,B 0,C 180,E1 -12319.751,E2 -12319.751} C_VEL
LIN {X 0,Y 374.88,Z 383.107,A -85,B 0,C 180,E1 -12321.374,E2 -12321.374} C_VEL
LIN {X 0,Y 374.668,Z 388.129,A -85,B 0,C 180,E1 -12322.997,E2 -12322.997} C_VEL
LIN {X 0,Y 374.579,Z 391.993,A -85,B 0,C 180,E1 -12324.617,E2 -12324.617} C_VEL
LIN {X 0,Y 374.585,Z 393.977,A -85,B 0,C 180,E1 -12325.696,E2 -12325.696} C_VEL
LIN {X 0,Y 374.567,Z 395.533,A -85,B 0,C 180,E1 -12326.773,E2 -12326.773} C_VEL
LIN {X 0,Y 374.67,Z 396.639,A -85,B 0,C 180,E1 -12327.85,E2 -12327.85} C_VEL
LIN {X 0,Y 374.667,Z 397.315,A -85,B 0,C 180,E1 -12328.925,E2 -12328.925} C_VEL
LIN {X 0,Y 374.656,Z 397.594,A -85,B 0,C 180,E1 -12330,E2 -12330} C_VEL
LIN {X 0,Y 374.656,Z 397.476,A -85,B 0,C 180,E1 -12331.075,E2 -12331.075} C_VEL
LIN {X 0,Y 374.628,Z 396.919,A -85,B 0,C 180,E1 -12332.15,E2 -12332.15} C_VEL
LIN {X 0,Y 374.576,Z 394.569,A -85,B 0,C 180,E1 -12334.304,E2 -12334.304} C_VEL
LIN {X 0,Y 374.549,Z 391.488,A -85,B 0,C 180,E1 -12336.016,E2 -12336.016} C_VEL
LIN {X 0,Y 374.722,Z 387.754,A -85,B 0,C 180,E1 -12337.544,E2 -12337.544} C_VEL
LIN {X 0,Y 375.003,Z 382.693,A -85,B 0,C 180,E1 -12339.166,E2 -12339.166} C_VEL
LIN {X 0,Y 375.469,Z 376.349,A -85,B 0,C 180,E1 -12340.788,E2 -12340.788} C_VEL
LIN {X 0,Y 376.297,Z 368.465,A -85,B 0,C 180,E1 -12342.403,E2 -12342.403} C_VEL
LIN {X 0,Y 377.29,Z 358.618,A -85,B 0,C 180,E1 -12344.014,E2 -12344.014} C_VEL
LIN {X 0,Y 378.281,Z 348.466,A -85,B 0,C 180,E1 -12345.352,E2 -12345.352} C_VEL
LIN {X 0,Y 379.374,Z 337.007,A -85,B 0,C 180,E1 -12346.548,E2 -12346.548} C_VEL
LIN {X 0,Y 380.447,Z 325.816,A -85,B 0,C 180,E1 -12347.469,E2 -12347.469} C_VEL
LIN {X 0,Y 381.461,Z 313.386,A -85,B 0,C 180,E1 -12348.252,E2 -12348.252} C_VEL
LIN {X 0,Y 382.346,Z 300.256,A -85,B 0,C 180,E1 -12348.833,E2 -12348.833} C_VEL
LIN {X 0,Y 382.877,Z 286.401,A -85,B 0,C 180,E1 -12349.223,E2 -12349.223} C_VEL
LIN {X 0,Y 383.993,Z 218.849,A -85,B 0,C 180,E1 -12350.58,E2 -12350.58} C_VEL
LIN {X 0,Y 381.071,Z 197.904,A -85,B 0,C 180,E1 -12351.215,E2 -12351.215} C_VEL
LIN {X 0,Y 378.358,Z 182.851,A -85,B 0,C 180,E1 -12351.735,E2 -12351.735} C_VEL
LIN {X 0,Y 379.906,Z 165.918,A -85,B 0,C 180,E1 -12355.181,E2 -12355.181} C_VEL
LIN {X 0,Y 380.102,Z 160.393,A -85,B 0,C 180,E1 -12356.343,E2 -12356.343} C_VEL
LIN {X 0,Y 377.724,Z 148.894,A -85,B 0,C 180,E1 -12359.015,E2 -12359.015} C_VEL
LIN {X 0,Y 375.965,Z 141.655,A -85,B 0,C 180,E1 -12360.832,E2 -12360.832} C_VEL
LIN {X 0,Y 375.981,Z 141.655,A -85,B 0,C 180,E1 -12364.667,E2 -12364.667} C_VEL
LIN {X 0,Y 375.978,Z 141.658,A -85,B 0,C 180,E1 -12368.271,E2 -12368.271} C_VEL
LIN {X 0,Y 375.961,Z 141.656,A -85,B 0,C 180,E1 -12371.605,E2 -12371.605} C_VEL
LIN {X 0,Y 375.927,Z 141.66,A -85,B 0,C 180,E1 -12375.268,E2 -12375.268} C_VEL
LIN {X 0,Y 375.96,Z 141.653,A -85,B 0,C 180,E1 -12378.394,E2 -12378.394} C_VEL
LIN {X 0,Y 375.977,Z 141.65,A -85,B 0,C 180,E1 -12381.728,E2 -12381.728} C_VEL
LIN {X 0,Y 375.979,Z 141.65,A -85,B 0,C 180,E1 -12385.332,E2 -12385.332} C_VEL
LIN {X 0,Y 375.957,Z 141.653,A -85,B 0,C 180,E1 -12388.438,E2 -12388.438} C_VEL
LIN {X 0,Y 375.995,Z 141.648,A -85,B 0,C 180,E1 -12392.141,E2 -12392.141} C_VEL
LIN {X 0,Y 376.004,Z 141.642,A -85,B 0,C 180,E1 -12394.539,E2 -12394.539} C_VEL
LIN {X 0,Y 375.956,Z 141.65,A -85,B 0,C 180,E1 -12398.045,E2 -12398.045} C_VEL
LIN {X 0,Y 376.023,Z 141.64,A -85,B 0,C 180,E1 -12401.474,E2 -12401.474} C_VEL
LIN {X 0,Y 376.057,Z 141.635,A -85,B 0,C 180,E1 -12404.832,E2 -12404.832} C_VEL
LIN {X 0,Y 376.048,Z 141.637,A -85,B 0,C 180,E1 -12408.136,E2 -12408.136} C_VEL
LIN {X 0,Y 376.256,Z 141.611,A -85,B 0,C 180,E1 -12411.877,E2 -12411.877} C_VEL
LIN {X 0,Y 376.17,Z 141.627,A -85,B 0,C 180,E1 -12414.64,E2 -12414.64} C_VEL
LIN {X 0,Y 376.352,Z 141.604,A -85,B 0,C 180,E1 -12417.859,E2 -12417.859} C_VEL
LIN {X 0,Y 376.487,Z 141.582,A -85,B 0,C 180,E1 -12420,E2 -12420} C_VEL
LIN {X 0,Y 376.187,Z 141.623,A -85,B 0,C 180,E1 -12423.213,E2 -12423.213} C_VEL
LIN {X 0,Y 376.227,Z 141.616,A -85,B 0,C 180,E1 -12426.538,E2 -12426.538} C_VEL
LIN {X 0,Y 376.117,Z 141.633,A -85,B 0,C 180,E1 -12429.681,E2 -12429.681} C_VEL
LIN {X 0,Y 376.087,Z 141.636,A -85,B 0,C 180,E1 -12433.657,E2 -12433.657} C_VEL
LIN {X 0,Y 376.042,Z 141.642,A -85,B 0,C 180,E1 -12437.607,E2 -12437.607} C_VEL
LIN {X 0,Y 375.976,Z 141.655,A -85,B 0,C 180,E1 -12440.832,E2 -12440.832} C_VEL
LIN {X 0,Y 375.992,Z 141.656,A -85,B 0,C 180,E1 -12444.281,E2 -12444.281} C_VEL
LIN {X 0,Y 376.017,Z 141.649,A -85,B 0,C 180,E1 -12446.652,E2 -12446.652} C_VEL
LIN {X 0,Y 376.004,Z 141.78,A -85,B 0,C 180,E1 -12449.768,E2 -12449.768} C_VEL
LIN {X 0,Y 377.227,Z 147.216,A -85,B 0,C 180,E1 -12451.255,E2 -12451.255} C_VEL
LIN {X 0,Y 383.827,Z 163.713,A -85,B 0,C 180,E1 -12452.073,E2 -12452.073} C_VEL
LIN {X 0,Y 384.966,Z 169.119,A -85,B 0,C 180,E1 -12452.264,E2 -12452.264} C_VEL
LIN {X 0,Y 383.231,Z 254.312,A -85,B 0,C 180,E1 -12453.993,E2 -12453.993} C_VEL
LIN {X 0,Y 382.731,Z 267.2,A -85,B 0,C 180,E1 -12454.457,E2 -12454.457} C_VEL
LIN {X 0,Y 382.176,Z 278.908,A -85,B 0,C 180,E1 -12455.076,E2 -12455.076} C_VEL
LIN {X 0,Y 381.348,Z 291.221,A -85,B 0,C 180,E1 -12455.948,E2 -12455.948} C_VEL
LIN {X 0,Y 380.424,Z 302.618,A -85,B 0,C 180,E1 -12457.004,E2 -12457.004} C_VEL
LIN {X 0,Y 379.399,Z 313.487,A -85,B 0,C 180,E1 -12458.268,E2 -12458.268} C_VEL
LIN {X 0,Y 378.416,Z 322.55,A -85,B 0,C 180,E1 -12459.58,E2 -12459.58} C_VEL
LIN {X 0,Y 377.469,Z 330.831,A -85,B 0,C 180,E1 -12461.057,E2 -12461.057} C_VEL
LIN {X 0,Y 376.556,Z 338.313,A -85,B 0,C 180,E1 -12462.712,E2 -12462.712} C_VEL
LIN {X 0,Y 376.009,Z 343.757,A -85,B 0,C 180,E1 -12464.223,E2 -12464.223} C_VEL
LIN {X 0,Y 375.401,Z 349.173,A -85,B 0,C 180,E1 -12466.157,E2 -12466.157} C_VEL
LIN {X 0,Y 375.083,Z 352.159,A -85,B 0,C 180,E1 -12467.582,E2 -12467.582} C_VEL
LIN {X 0,Y 374.794,Z 354.311,A -85,B 0,C 180,E1 -12468.982,E2 -12468.982} C_VEL
LIN {X 0,Y 374.628,Z 355.772,A -85,B 0,C 180,E1 -12470.37,E2 -12470.37} C_VEL
LIN {X 0,Y 374.524,Z 356.625,A -85,B 0,C 180,E1 -12472.011,E2 -12472.011} C_VEL
LIN {X 0,Y 374.51,Z 356.483,A -85,B 0,C 180,E1 -12473.797,E2 -12473.797} C_VEL
LIN {X 0,Y 374.602,Z 355.06,A -85,B 0,C 180,E1 -12475.748,E2 -12475.748} C_VEL
LIN {X 0,Y 374.84,Z 352.582,A -85,B 0,C 180,E1 -12477.535,E2 -12477.535} C_VEL
LIN {X 0,Y 375.193,Z 348.179,A -85,B 0,C 180,E1 -12479.619,E2 -12479.619} C_VEL
LIN {X 0,Y 375.686,Z 342.414,A -85,B 0,C 180,E1 -12481.55,E2 -12481.55} C_VEL
LIN {X 0,Y 376.371,Z 335.306,A -85,B 0,C 180,E1 -12483.375,E2 -12483.375} C_VEL
LIN {X 0,Y 377.042,Z 327.734,A -85,B 0,C 180,E1 -12484.91,E2 -12484.91} C_VEL
LIN {X 0,Y 377.919,Z 318.424,A -85,B 0,C 180,E1 -12486.433,E2 -12486.433} C_VEL
LIN {X 0,Y 378.725,Z 308.712,A -85,B 0,C 180,E1 -12487.721,E2 -12487.721} C_VEL
LIN {X 0,Y 379.569,Z 298.233,A -85,B 0,C 180,E1 -12488.835,E2 -12488.835} C_VEL
LIN {X 0,Y 380.328,Z 286.871,A -85,B 0,C 180,E1 -12489.799,E2 -12489.799} C_VEL
LIN {X 0,Y 380.987,Z 274.497,A -85,B 0,C 180,E1 -12490.607,E2 -12490.607} C_VEL
LIN {X 0,Y 381.497,Z 261.959,A -85,B 0,C 180,E1 -12491.193,E2 -12491.193} C_VEL
LIN {X 0,Y 381.853,Z 248.576,A -85,B 0,C 180,E1 -12491.593,E2 -12491.593} C_VEL
LIN {X 0,Y 383.25,Z 168.129,A -85,B 0,C 180,E1 -12493.179,E2 -12493.179} C_VEL
LIN {X 0,Y 380.877,Z 157.42,A -85,B 0,C 180,E1 -12493.521,E2 -12493.521} C_VEL
LIN {X 0,Y 376.857,Z 145.658,A -85,B 0,C 180,E1 -12493.999,E2 -12493.999} C_VEL
LIN {X 0,Y 376.104,Z 141.638,A -85,B 0,C 180,E1 -12495.112,E2 -12495.112} C_VEL
LIN {X 0,Y 376.046,Z 141.641,A -85,B 0,C 180,E1 -12498.137,E2 -12498.137} C_VEL
LIN {X 0,Y 376.218,Z 141.621,A -85,B 0,C 180,E1 -12501.919,E2 -12501.919} C_VEL
LIN {X 0,Y 376.168,Z 141.624,A -85,B 0,C 180,E1 -12504.64,E2 -12504.64} C_VEL
LIN {X 0,Y 376.351,Z 141.603,A -85,B 0,C 180,E1 -12507.86,E2 -12507.86} C_VEL
LIN {X 0,Y 376.319,Z 141.606,A -85,B 0,C 180,E1 -12509.203,E2 -12509.203} C_VEL
LIN {X 0,Y 375.745,Z 141.678,A -85,B 0,C 180,E1 -12510.097,E2 -12510.097} C_VEL
LIN {X 0,Y 372.848,Z 142.042,A -85,B 0,C 180,E1 -12511.549,E2 -12511.549} C_VEL
LIN {X 0,Y 370.292,Z 142.36,A -85,B 0,C 180,E1 -12512.723,E2 -12512.723} C_VEL
LIN {X 0,Y 369.143,Z 142.503,A -85,B 0,C 180,E1 -12513.633,E2 -12513.633} C_VEL
LIN {X 0,Y 369.026,Z 142.515,A -85,B 0,C 180,E1 -12513.942,E2 -12513.942} C_VEL
LIN {X 0,Y 369.174,Z 142.497,A -85,B 0,C 180,E1 -12516.559,E2 -12516.559} C_VEL
LIN {X 0,Y 369.063,Z 142.51,A -85,B 0,C 180,E1 -12519.868,E2 -12519.868} C_VEL
LIN {X 0,Y 369.037,Z 142.513,A -85,B 0,C 180,E1 -12523.772,E2 -12523.772} C_VEL
LIN {X 0,Y 368.99,Z 142.519,A -85,B 0,C 180,E1 -12527.743,E2 -12527.743} C_VEL
LIN {X 0,Y 368.909,Z 142.531,A -85,B 0,C 180,E1 -12531.221,E2 -12531.221} C_VEL
LIN {X 0,Y 368.955,Z 142.529,A -85,B 0,C 180,E1 -12534.775,E2 -12534.775} C_VEL
LIN {X 0,Y 368.967,Z 142.523,A -85,B 0,C 180,E1 -12537.203,E2 -12537.203} C_VEL
LIN {X 0,Y 368.918,Z 142.527,A -85,B 0,C 180,E1 -12539.69,E2 -12539.69} C_VEL
LIN {X 0,Y 368.896,Z 142.532,A -85,B 0,C 180,E1 -12543.043,E2 -12543.043} C_VEL
LIN {X 0,Y 368.915,Z 142.532,A -85,B 0,C 180,E1 -12546.197,E2 -12546.197} C_VEL
LIN {X 0,Y 368.9,Z 142.531,A -85,B 0,C 180,E1 -12548.953,E2 -12548.953} C_VEL
LIN {X 0,Y 368.88,Z 142.536,A -85,B 0,C 180,E1 -12552.009,E2 -12552.009} C_VEL
LIN {X 0,Y 368.879,Z 142.532,A -85,B 0,C 180,E1 -12555.176,E2 -12555.176} C_VEL
LIN {X 0,Y 368.882,Z 142.538,A -85,B 0,C 180,E1 -12558.178,E2 -12558.178} C_VEL
LIN {X 0,Y 368.909,Z 142.529,A -85,B 0,C 180,E1 -12561.359,E2 -12561.359} C_VEL
LIN {X 0,Y 368.935,Z 142.525,A -85,B 0,C 180,E1 -12565.147,E2 -12565.147} C_VEL
LIN {X 0,Y 368.927,Z 142.526,A -85,B 0,C 180,E1 -12569.047,E2 -12569.047} C_VEL
LIN {X 0,Y 368.978,Z 142.524,A -85,B 0,C 180,E1 -12571.564,E2 -12571.564} C_VEL
LIN {X 0,Y 368.998,Z 142.521,A -85,B 0,C 180,E1 -12574.02,E2 -12574.02} C_VEL
LIN {X 0,Y 368.921,Z 142.533,A -85,B 0,C 180,E1 -12577.604,E2 -12577.604} C_VEL
LIN {X 0,Y 368.982,Z 142.521,A -85,B 0,C 180,E1 -12581.107,E2 -12581.107} C_VEL
LIN {X 0,Y 368.996,Z 142.518,A -85,B 0,C 180,E1 -12584.535,E2 -12584.535} C_VEL
LIN {X 0,Y 369.004,Z 142.518,A -85,B 0,C 180,E1 -12587.907,E2 -12587.907} C_VEL
LIN {X 0,Y 369.228,Z 142.491,A -85,B 0,C 180,E1 -12591.801,E2 -12591.801} C_VEL
LIN {X 0,Y 369.143,Z 142.5,A -85,B 0,C 180,E1 -12594.538,E2 -12594.538} C_VEL
LIN {X 0,Y 369.317,Z 142.478,A -85,B 0,C 180,E1 -12597.819,E2 -12597.819} C_VEL
LIN {X 0,Y 369.457,Z 142.46,A -85,B 0,C 180,E1 -12600,E2 -12600} C_VEL
LIN {X 0,Y 369.317,Z 142.478,A -85,B 0,C 180,E1 -12602.181,E2 -12602.181} C_VEL
LIN {X 0,Y 369.197,Z 142.495,A -85,B 0,C 180,E1 -12606.559,E2 -12606.559} C_VEL
LIN {X 0,Y 369.121,Z 142.507,A -85,B 0,C 180,E1 -12608.762,E2 -12608.762} C_VEL
LIN {X 0,Y 369.004,Z 142.517,A -85,B 0,C 180,E1 -12612.094,E2 -12612.094} C_VEL
LIN {X 0,Y 368.997,Z 142.518,A -85,B 0,C 180,E1 -12615.465,E2 -12615.465} C_VEL
LIN {X 0,Y 368.982,Z 142.523,A -85,B 0,C 180,E1 -12618.893,E2 -12618.893} C_VEL
LIN {X 0,Y 368.924,Z 142.531,A -85,B 0,C 180,E1 -12622.396,E2 -12622.396} C_VEL
LIN {X 0,Y 368.999,Z 142.519,A -85,B 0,C 180,E1 -12625.98,E2 -12625.98} C_VEL
LIN {X 0,Y 368.961,Z 142.524,A -85,B 0,C 180,E1 -12628.812,E2 -12628.812} C_VEL
LIN {X 0,Y 368.898,Z 142.536,A -85,B 0,C 180,E1 -12632.238,E2 -12632.238} C_VEL
LIN {X 0,Y 368.929,Z 142.526,A -85,B 0,C 180,E1 -12635.002,E2 -12635.002} C_VEL
LIN {X 0,Y 368.913,Z 142.53,A -85,B 0,C 180,E1 -12638.641,E2 -12638.641} C_VEL
LIN {X 0,Y 368.911,Z 142.532,A -85,B 0,C 180,E1 -12641.819,E2 -12641.819} C_VEL
LIN {X 0,Y 368.881,Z 142.532,A -85,B 0,C 180,E1 -12645.176,E2 -12645.176} C_VEL
LIN {X 0,Y 368.911,Z 142.532,A -85,B 0,C 180,E1 -12648.182,E2 -12648.182} C_VEL
LIN {X 0,Y 368.914,Z 142.53,A -85,B 0,C 180,E1 -12651.359,E2 -12651.359} C_VEL
LIN {X 0,Y 368.938,Z 142.526,A -85,B 0,C 180,E1 -12655.147,E2 -12655.147} C_VEL
LIN {X 0,Y 368.931,Z 142.528,A -85,B 0,C 180,E1 -12659.047,E2 -12659.047} C_VEL
LIN {X 0,Y 368.963,Z 142.753,A -85,B 0,C 180,E1 -12659.605,E2 -12659.605} C_VEL
LIN {X 0,Y 371.804,Z 155.813,A -85,B 0,C 180,E1 -12662.675,E2 -12662.675} C_VEL
LIN {X 0,Y 372.795,Z 161.696,A -85,B 0,C 180,E1 -12664.004,E2 -12664.004} C_VEL
LIN {X 0,Y 371.542,Z 176.923,A -85,B 0,C 180,E1 -12667.184,E2 -12667.184} C_VEL
LIN {X 0,Y 371.03,Z 184.474,A -85,B 0,C 180,E1 -12668.732,E2 -12668.732} C_VEL
LIN {X 0,Y 375.856,Z 220.565,A -85,B 0,C 180,E1 -12669.743,E2 -12669.743} C_VEL
LIN {X 0,Y 374.656,Z 293.256,A -85,B 0,C 180,E1 -12671.227,E2 -12671.227} C_VEL
LIN {X 0,Y 374.019,Z 306.303,A -85,B 0,C 180,E1 -12671.69,E2 -12671.69} C_VEL
LIN {X 0,Y 373.126,Z 319.53,A -85,B 0,C 180,E1 -12672.39,E2 -12672.39} C_VEL
LIN {X 0,Y 372.17,Z 331.497,A -85,B 0,C 180,E1 -12673.263,E2 -12673.263} C_VEL
LIN {X 0,Y 371.123,Z 342.993,A -85,B 0,C 180,E1 -12674.345,E2 -12674.345} C_VEL
LIN {X 0,Y 370.242,Z 353.409,A -85,B 0,C 180,E1 -12675.577,E2 -12675.577} C_VEL
LIN {X 0,Y 369.313,Z 363.531,A -85,B 0,C 180,E1 -12677.079,E2 -12677.079} C_VEL
LIN {X 0,Y 368.497,Z 372.45,A -85,B 0,C 180,E1 -12678.727,E2 -12678.727} C_VEL
LIN {X 0,Y 368.009,Z 379.581,A -85,B 0,C 180,E1 -12680.381,E2 -12680.381} C_VEL
LIN {X 0,Y 367.672,Z 386.087,A -85,B 0,C 180,E1 -12682.311,E2 -12682.311} C_VEL
LIN {X 0,Y 367.489,Z 390.377,A -85,B 0,C 180,E1 -12683.973,E2 -12683.973} C_VEL
LIN {X 0,Y 367.51,Z 393.529,A -85,B 0,C 180,E1 -12685.613,E2 -12685.613} C_VEL
LIN {X 0,Y 367.477,Z 395.096,A -85,B 0,C 180,E1 -12686.711,E2 -12686.711} C_VEL
LIN {X 0,Y 367.571,Z 396.223,A -85,B 0,C 180,E1 -12687.808,E2 -12687.808} C_VEL
LIN {X 0,Y 367.6,Z 396.911,A -85,B 0,C 180,E1 -12688.904,E2 -12688.904} C_VEL
LIN {X 0,Y 367.587,Z 397.199,A -85,B 0,C 180,E1 -12690,E2 -12690} C_VEL
LIN {X 0,Y 367.589,Z 397.092,A -85,B 0,C 180,E1 -12691.095,E2 -12691.095} C_VEL
LIN {X 0,Y 367.528,Z 396.553,A -85,B 0,C 180,E1 -12692.192,E2 -12692.192} C_VEL
LIN {X 0,Y 367.5,Z 394.224,A -85,B 0,C 180,E1 -12694.387,E2 -12694.387} C_VEL
LIN {X 0,Y 367.471,Z 391.428,A -85,B 0,C 180,E1 -12696.001,E2 -12696.001} C_VEL
LIN {X 0,Y 367.661,Z 387.449,A -85,B 0,C 180,E1 -12697.69,E2 -12697.69} C_VEL
LIN {X 0,Y 367.95,Z 382.409,A -85,B 0,C 180,E1 -12699.343,E2 -12699.343} C_VEL
LIN {X 0,Y 368.459,Z 376.088,A -85,B 0,C 180,E1 -12700.996,E2 -12700.996} C_VEL
LIN {X 0,Y 369.34,Z 368.247,A -85,B 0,C 180,E1 -12702.64,E2 -12702.64} C_VEL
LIN {X 0,Y 370.384,Z 358.431,A -85,B 0,C 180,E1 -12704.281,E2 -12704.281} C_VEL
LIN {X 0,Y 371.406,Z 348.339,A -85,B 0,C 180,E1 -12705.643,E2 -12705.643} C_VEL
LIN {X 0,Y 372.577,Z 336.982,A -85,B 0,C 180,E1 -12706.859,E2 -12706.859} C_VEL
LIN {X 0,Y 373.676,Z 325.907,A -85,B 0,C 180,E1 -12707.796,E2 -12707.796} C_VEL
LIN {X 0,Y 374.755,Z 313.69,A -85,B 0,C 180,E1 -12708.591,E2 -12708.591} C_VEL
LIN {X 0,Y 375.667,Z 300.955,A -85,B 0,C 180,E1 -12709.181,E2 -12709.181} C_VEL
LIN {X 0,Y 376.211,Z 287.833,A -85,B 0,C 180,E1 -12709.578,E2 -12709.578} C_VEL
LIN {X 0,Y 377.432,Z 219.434,A -85,B 0,C 180,E1 -12710.983,E2 -12710.983} C_VEL
LIN {X 0,Y 374.21,Z 196.714,A -85,B 0,C 180,E1 -12711.694,E2 -12711.694} C_VEL
LIN {X 0,Y 371.597,Z 182.335,A -85,B 0,C 180,E1 -12712.226,E2 -12712.226} C_VEL
LIN {X 0,Y 373.17,Z 165.79,A -85,B 0,C 180,E1 -12715.668,E2 -12715.668} C_VEL
LIN {X 0,Y 373.178,Z 161.642,A -85,B 0,C 180,E1 -12716.569,E2 -12716.569} C_VEL
LIN {X 0,Y 370.983,Z 151.07,A -85,B 0,C 180,E1 -12719.082,E2 -12719.082} C_VEL
LIN {X 0,Y 368.933,Z 142.53,A -85,B 0,C 180,E1 -12721.271,E2 -12721.271} C_VEL
LIN {X 0,Y 368.93,Z 142.531,A -85,B 0,C 180,E1 -12725.001,E2 -12725.001} C_VEL
LIN {X 0,Y 368.913,Z 142.535,A -85,B 0,C 180,E1 -12728.641,E2 -12728.641} C_VEL
LIN {X 0,Y 368.911,Z 142.536,A -85,B 0,C 180,E1 -12731.818,E2 -12731.818} C_VEL
LIN {X 0,Y 368.88,Z 142.538,A -85,B 0,C 180,E1 -12735.175,E2 -12735.175} C_VEL
LIN {X 0,Y 368.91,Z 142.531,A -85,B 0,C 180,E1 -12738.181,E2 -12738.181} C_VEL
LIN {X 0,Y 368.912,Z 142.528,A -85,B 0,C 180,E1 -12741.358,E2 -12741.358} C_VEL
LIN {X 0,Y 368.936,Z 142.527,A -85,B 0,C 180,E1 -12745.146,E2 -12745.146} C_VEL
LIN {X 0,Y 368.928,Z 142.529,A -85,B 0,C 180,E1 -12749.046,E2 -12749.046} C_VEL
LIN {X 0,Y 368.979,Z 142.521,A -85,B 0,C 180,E1 -12751.564,E2 -12751.564} C_VEL
LIN {X 0,Y 368.998,Z 142.515,A -85,B 0,C 180,E1 -12754.019,E2 -12754.019} C_VEL
LIN {X 0,Y 368.923,Z 142.524,A -85,B 0,C 180,E1 -12757.604,E2 -12757.604} C_VEL
LIN {X 0,Y 368.981,Z 142.516,A -85,B 0,C 180,E1 -12761.107,E2 -12761.107} C_VEL
LIN {X 0,Y 368.996,Z 142.514,A -85,B 0,C 180,E1 -12764.535,E2 -12764.535} C_VEL
LIN {X 0,Y 369.003,Z 142.515,A -85,B 0,C 180,E1 -12767.906,E2 -12767.906} C_VEL
LIN {X 0,Y 369.228,Z 142.487,A -85,B 0,C 180,E1 -12771.8,E2 -12771.8} C_VEL
LIN {X 0,Y 369.143,Z 142.502,A -85,B 0,C 180,E1 -12774.537,E2 -12774.537} C_VEL
LIN {X 0,Y 369.317,Z 142.48,A -85,B 0,C 180,E1 -12777.819,E2 -12777.819} C_VEL
LIN {X 0,Y 369.457,Z 142.458,A -85,B 0,C 180,E1 -12780,E2 -12780} C_VEL
LIN {X 0,Y 369.317,Z 142.479,A -85,B 0,C 180,E1 -12782.181,E2 -12782.181} C_VEL
LIN {X 0,Y 369.197,Z 142.493,A -85,B 0,C 180,E1 -12786.558,E2 -12786.558} C_VEL
LIN {X 0,Y 369.065,Z 142.512,A -85,B 0,C 180,E1 -12789.868,E2 -12789.868} C_VEL
LIN {X 0,Y 369.035,Z 142.514,A -85,B 0,C 180,E1 -12793.772,E2 -12793.772} C_VEL
LIN {X 0,Y 368.999,Z 142.52,A -85,B 0,C 180,E1 -12797.768,E2 -12797.768} C_VEL
LIN {X 0,Y 368.927,Z 142.53,A -85,B 0,C 180,E1 -12801.22,E2 -12801.22} C_VEL
LIN {X 0,Y 368.955,Z 142.534,A -85,B 0,C 180,E1 -12804.775,E2 -12804.775} C_VEL
LIN {X 0,Y 368.961,Z 142.53,A -85,B 0,C 180,E1 -12807.203,E2 -12807.203} C_VEL
LIN {X 0,Y 368.935,Z 142.55,A -85,B 0,C 180,E1 -12809.318,E2 -12809.318} C_VEL
LIN {X 0,Y 370.146,Z 147.746,A -85,B 0,C 180,E1 -12810.761,E2 -12810.761} C_VEL
LIN {X 0,Y 377.652,Z 166.299,A -85,B 0,C 180,E1 -12811.716,E2 -12811.716} C_VEL
LIN {X 0,Y 378.444,Z 169.745,A -85,B 0,C 180,E1 -12811.845,E2 -12811.845} C_VEL
LIN {X 0,Y 376.619,Z 255.154,A -85,B 0,C 180,E1 -12813.616,E2 -12813.616} C_VEL
LIN {X 0,Y 376.094,Z 268.096,A -85,B 0,C 180,E1 -12814.097,E2 -12814.097} C_VEL
LIN {X 0,Y 375.493,Z 280.417,A -85,B 0,C 180,E1 -12814.773,E2 -12814.773} C_VEL
LIN {X 0,Y 374.554,Z 292.876,A -85,B 0,C 180,E1 -12815.698,E2 -12815.698} C_VEL
LIN {X 0,Y 373.591,Z 304.106,A -85,B 0,C 180,E1 -12816.78,E2 -12816.78} C_VEL
LIN {X 0,Y 372.541,Z 314.589,A -85,B 0,C 180,E1 -12818.046,E2 -12818.046} C_VEL
LIN {X 0,Y 371.47,Z 323.761,A -85,B 0,C 180,E1 -12819.426,E2 -12819.426} C_VEL
LIN {X 0,Y 370.483,Z 331.956,A -85,B 0,C 180,E1 -12820.943,E2 -12820.943} C_VEL
LIN {X 0,Y 369.626,Z 338.604,A -85,B 0,C 180,E1 -12822.453,E2 -12822.453} C_VEL
LIN {X 0,Y 368.92,Z 345.057,A -85,B 0,C 180,E1 -12824.303,E2 -12824.303} C_VEL
LIN {X 0,Y 368.434,Z 349.272,A -85,B 0,C 180,E1 -12825.858,E2 -12825.858} C_VEL
LIN {X 0,Y 368.07,Z 352.336,A -85,B 0,C 180,E1 -12827.325,E2 -12827.325} C_VEL
LIN {X 0,Y 367.642,Z 355.409,A -85,B 0,C 180,E1 -12829.462,E2 -12829.462} C_VEL
LIN {X 0,Y 367.469,Z 356.919,A -85,B 0,C 180,E1 -12831.641,E2 -12831.641} C_VEL
LIN {X 0,Y 367.434,Z 356.934,A -85,B 0,C 180,E1 -12833.634,E2 -12833.634} C_VEL
LIN {X 0,Y 367.476,Z 355.898,A -85,B 0,C 180,E1 -12835.323,E2 -12835.323} C_VEL
LIN {X 0,Y 367.706,Z 353.529,A -85,B 0,C 180,E1 -12837.243,E2 -12837.243} C_VEL
LIN {X 0,Y 368.053,Z 349.67,A -85,B 0,C 180,E1 -12839.235,E2 -12839.235} C_VEL
LIN {X 0,Y 368.427,Z 345.476,A -85,B 0,C 180,E1 -12840.824,E2 -12840.824} C_VEL
LIN {X 0,Y 368.919,Z 339.893,A -85,B 0,C 180,E1 -12842.486,E2 -12842.486} C_VEL
LIN {X 0,Y 369.554,Z 333.28,A -85,B 0,C 180,E1 -12844.062,E2 -12844.062} C_VEL
LIN {X 0,Y 370.402,Z 324.553,A -85,B 0,C 180,E1 -12845.728,E2 -12845.728} C_VEL
LIN {X 0,Y 371.281,Z 315.149,A -85,B 0,C 180,E1 -12847.167,E2 -12847.167} C_VEL
LIN {X 0,Y 372.113,Z 305.332,A -85,B 0,C 180,E1 -12848.39,E2 -12848.39} C_VEL
LIN {X 0,Y 373,Z 294.688,A -85,B 0,C 180,E1 -12849.457,E2 -12849.457} C_VEL
LIN {X 0,Y 373.812,Z 282.154,A -85,B 0,C 180,E1 -12850.434,E2 -12850.434} C_VEL
LIN {X 0,Y 374.365,Z 270.841,A -85,B 0,C 180,E1 -12851.105,E2 -12851.105} C_VEL
LIN {X 0,Y 374.826,Z 258.08,A -85,B 0,C 180,E1 -12851.646,E2 -12851.646} C_VEL
LIN {X 0,Y 375.223,Z 242.128,A -85,B 0,C 180,E1 -12852.035,E2 -12852.035} C_VEL
LIN {X 0,Y 376.472,Z 168.734,A -85,B 0,C 180,E1 -12853.51,E2 -12853.51} C_VEL
LIN {X 0,Y 374.376,Z 159.552,A -85,B 0,C 180,E1 -12853.815,E2 -12853.815} C_VEL
LIN {X 0,Y 369.727,Z 146.024,A -85,B 0,C 180,E1 -12854.376,E2 -12854.376} C_VEL
LIN {X 0,Y 369.052,Z 142.516,A -85,B 0,C 180,E1 -12855.35,E2 -12855.35} C_VEL
LIN {X 0,Y 369.002,Z 142.521,A -85,B 0,C 180,E1 -12857.907,E2 -12857.907} C_VEL
LIN {X 0,Y 369.165,Z 142.5,A -85,B 0,C 180,E1 -12861.87,E2 -12861.87} C_VEL
LIN {X 0,Y 369.141,Z 142.5,A -85,B 0,C 180,E1 -12864.538,E2 -12864.538} C_VEL
LIN {X 0,Y 369.316,Z 142.48,A -85,B 0,C 180,E1 -12867.819,E2 -12867.819} C_VEL
LIN {X 0,Y 369.457,Z 142.461,A -85,B 0,C 180,E1 -12870,E2 -12870} C_VEL
LIN {X 0,Y 369.317,Z 142.478,A -85,B 0,C 180,E1 -12872.181,E2 -12872.181} C_VEL
LIN {X 0,Y 369.026,Z 142.515,A -85,B 0,C 180,E1 -12873.942,E2 -12873.942} C_VEL
LIN {X 0,Y 368.31,Z 142.608,A -85,B 0,C 180,E1 -12874.854,E2 -12874.854} C_VEL
LIN {X 0,Y 365.495,Z 142.954,A -85,B 0,C 180,E1 -12876.338,E2 -12876.338} C_VEL
LIN {X 0,Y 363.145,Z 143.249,A -85,B 0,C 180,E1 -12877.538,E2 -12877.538} C_VEL
LIN {X 0,Y 362.134,Z 143.374,A -85,B 0,C 180,E1 -12878.465,E2 -12878.465} C_VEL
LIN {X 0,Y 362.048,Z 143.386,A -85,B 0,C 180,E1 -12878.779,E2 -12878.779} C_VEL
LIN {X 0,Y 361.959,Z 143.395,A -85,B 0,C 180,E1 -12882.332,E2 -12882.332} C_VEL
LIN {X 0,Y 361.961,Z 143.397,A -85,B 0,C 180,E1 -12884.62,E2 -12884.62} C_VEL
LIN {X 0,Y 361.91,Z 143.401,A -85,B 0,C 180,E1 -12888.102,E2 -12888.102} C_VEL
LIN {X 0,Y 361.861,Z 143.407,A -85,B 0,C 180,E1 -12891.655,E2 -12891.655} C_VEL
LIN {X 0,Y 361.926,Z 143.4,A -85,B 0,C 180,E1 -12895.29,E2 -12895.29} C_VEL
LIN {X 0,Y 361.918,Z 143.4,A -85,B 0,C 180,E1 -12897.778,E2 -12897.778} C_VEL
LIN {X 0,Y 361.845,Z 143.409,A -85,B 0,C 180,E1 -12901.285,E2 -12901.285} C_VEL
LIN {X 0,Y 361.853,Z 143.412,A -85,B 0,C 180,E1 -12904.28,E2 -12904.28} C_VEL
LIN {X 0,Y 361.861,Z 143.407,A -85,B 0,C 180,E1 -12907.223,E2 -12907.223} C_VEL
LIN {X 0,Y 361.834,Z 143.412,A -85,B 0,C 180,E1 -12910.755,E2 -12910.755} C_VEL
LIN {X 0,Y 361.816,Z 143.417,A -85,B 0,C 180,E1 -12914.368,E2 -12914.368} C_VEL
LIN {X 0,Y 361.835,Z 143.411,A -85,B 0,C 180,E1 -12917.568,E2 -12917.568} C_VEL
LIN {X 0,Y 361.869,Z 143.406,A -85,B 0,C 180,E1 -12920.973,E2 -12920.973} C_VEL
LIN {X 0,Y 361.873,Z 143.406,A -85,B 0,C 180,E1 -12924.655,E2 -12924.655} C_VEL
LIN {X 0,Y 361.836,Z 143.411,A -85,B 0,C 180,E1 -12928.371,E2 -12928.371} C_VEL
LIN {X 0,Y 361.899,Z 143.402,A -85,B 0,C 180,E1 -12930.955,E2 -12930.955} C_VEL
LIN {X 0,Y 361.953,Z 143.398,A -85,B 0,C 180,E1 -12933.475,E2 -12933.475} C_VEL
LIN {X 0,Y 361.878,Z 143.406,A -85,B 0,C 180,E1 -12937.144,E2 -12937.144} C_VEL
LIN {X 0,Y 361.92,Z 143.399,A -85,B 0,C 180,E1 -12940.724,E2 -12940.724} C_VEL
LIN {X 0,Y 361.945,Z 143.397,A -85,B 0,C 180,E1 -12944.226,E2 -12944.226} C_VEL
LIN {X 0,Y 361.997,Z 143.39,A -85,B 0,C 180,E1 -12946.528,E2 -12946.528} C_VEL
LIN {X 0,Y 362.03,Z 143.387,A -85,B 0,C 180,E1 -12949.938,E2 -12949.938} C_VEL
LIN {X 0,Y 362.15,Z 143.371,A -85,B 0,C 180,E1 -12952.193,E2 -12952.193} C_VEL
LIN {X 0,Y 362.117,Z 143.375,A -85,B 0,C 180,E1 -12954.431,E2 -12954.431} C_VEL
LIN {X 0,Y 362.281,Z 143.355,A -85,B 0,C 180,E1 -12957.777,E2 -12957.777} C_VEL
LIN {X 0,Y 362.427,Z 143.336,A -85,B 0,C 180,E1 -12960,E2 -12960} C_VEL
LIN {X 0,Y 362.281,Z 143.354,A -85,B 0,C 180,E1 -12962.224,E2 -12962.224} C_VEL
LIN {X 0,Y 362.159,Z 143.373,A -85,B 0,C 180,E1 -12966.687,E2 -12966.687} C_VEL
LIN {X 0,Y 362.03,Z 143.386,A -85,B 0,C 180,E1 -12970.062,E2 -12970.062} C_VEL
LIN {X 0,Y 361.997,Z 143.39,A -85,B 0,C 180,E1 -12973.899,E2 -12973.899} C_VEL
LIN {X 0,Y 361.967,Z 143.394,A -85,B 0,C 180,E1 -12977.939,E2 -12977.939} C_VEL
LIN {X 0,Y 361.861,Z 143.407,A -85,B 0,C 180,E1 -12981.655,E2 -12981.655} C_VEL
LIN {X 0,Y 361.927,Z 143.399,A -85,B 0,C 180,E1 -12985.29,E2 -12985.29} C_VEL
LIN {X 0,Y 361.918,Z 143.4,A -85,B 0,C 180,E1 -12987.779,E2 -12987.779} C_VEL
LIN {X 0,Y 361.846,Z 143.408,A -85,B 0,C 180,E1 -12991.286,E2 -12991.286} C_VEL
LIN {X 0,Y 361.854,Z 143.413,A -85,B 0,C 180,E1 -12994.281,E2 -12994.281} C_VEL
LIN {X 0,Y 361.866,Z 143.406,A -85,B 0,C 180,E1 -12997.224,E2 -12997.224} C_VEL
LIN {X 0,Y 361.873,Z 143.406,A -85,B 0,C 180,E1 -13000.763,E2 -13000.763} C_VEL
LIN {X 0,Y 361.823,Z 143.414,A -85,B 0,C 180,E1 -13004.368,E2 -13004.368} C_VEL
LIN {X 0,Y 361.857,Z 143.41,A -85,B 0,C 180,E1 -13007.565,E2 -13007.565} C_VEL
LIN {X 0,Y 361.875,Z 143.405,A -85,B 0,C 180,E1 -13010.973,E2 -13010.973} C_VEL
LIN {X 0,Y 361.876,Z 143.405,A -85,B 0,C 180,E1 -13014.655,E2 -13014.655} C_VEL
LIN {X 0,Y 361.839,Z 143.41,A -85,B 0,C 180,E1 -13018.371,E2 -13018.371} C_VEL
LIN {X 0,Y 361.922,Z 143.578,A -85,B 0,C 180,E1 -13019.295,E2 -13019.295} C_VEL
LIN {X 0,Y 364.785,Z 156.779,A -85,B 0,C 180,E1 -13022.459,E2 -13022.459} C_VEL
